// TIA Portal V17 export
// export: Created 2024-08-26T21:07:18.1732783Z, ExportSetting WithDefaults, DisplayName Totally Integrated Automation Portal, DisplayVersion V17 Update 7, DisplayName TIA Portal Openness, DisplayVersion V17 Update 7, DisplayName TIA Portal Version Control Interface, DisplayVersion V17, DisplayName SINAMICS Startdrive Advanced, DisplayVersion V17 SP2, DisplayName SINAMICS Startdrive G110M, G120, G120C, G120D, G120P, G115D, DisplayVersion V17 SP2, DisplayName SINAMICS Startdrive G130, G150, S120, S150, SINAMICS MV, S210, DisplayVersion V17 SP2, DisplayName STEP 7 Professional, DisplayVersion V17 Update 7, DisplayName STEP 7 Safety, DisplayVersion V17 Update 6, DisplayName WinCC Advanced / Unified PC, DisplayVersion V17 Update 7
FUNCTION "hmiControl" : Void   // FC3, LAD
{ S7_Optimized_Access := 'TRUE' }
VERSION : 0.1
// stored: AutoNumber true, IsIECCheckEnabled false, SetENOAutomatically false, UDAEnableTagReadback false
   VAR_TEMP   // added for the SCL form of the ladder/FBD networks
      _w1 : Bool;
      _w2 : Bool;
      _w3 : Bool;
      _w4 : Bool;
      _w5 : Bool;
      _w6 : Bool;
      _w7 : Bool;
      _w8 : Bool;
      _w9 : Bool;
      _w10 : Bool;
      _w11 : Bool;
      _w12 : Bool;
      _w13 : Bool;
      _w14 : Bool;
      _w15 : Bool;
      _w16 : Bool;
      _w17 : Bool;
      _w18 : Bool;
      _w19 : Bool;
      _w20 : Bool;
      _w21 : Bool;
      _w22 : Bool;
      _w23 : Bool;
      _w24 : Bool;
      _w25 : Bool;
      _w26 : Bool;
      _w27 : Bool;
      _w28 : Bool;
      _w29 : Bool;
      _w30 : Bool;
      _w31 : Bool;
      _w32 : Bool;
   END_VAR
BEGIN

REGION Network 1: VISUALIZACIÓN DE MODELOS: SI CADA MODELO TIENE UN NOMBRE GRABADO, SE ACTIVA SU VISUALIZACIÓN
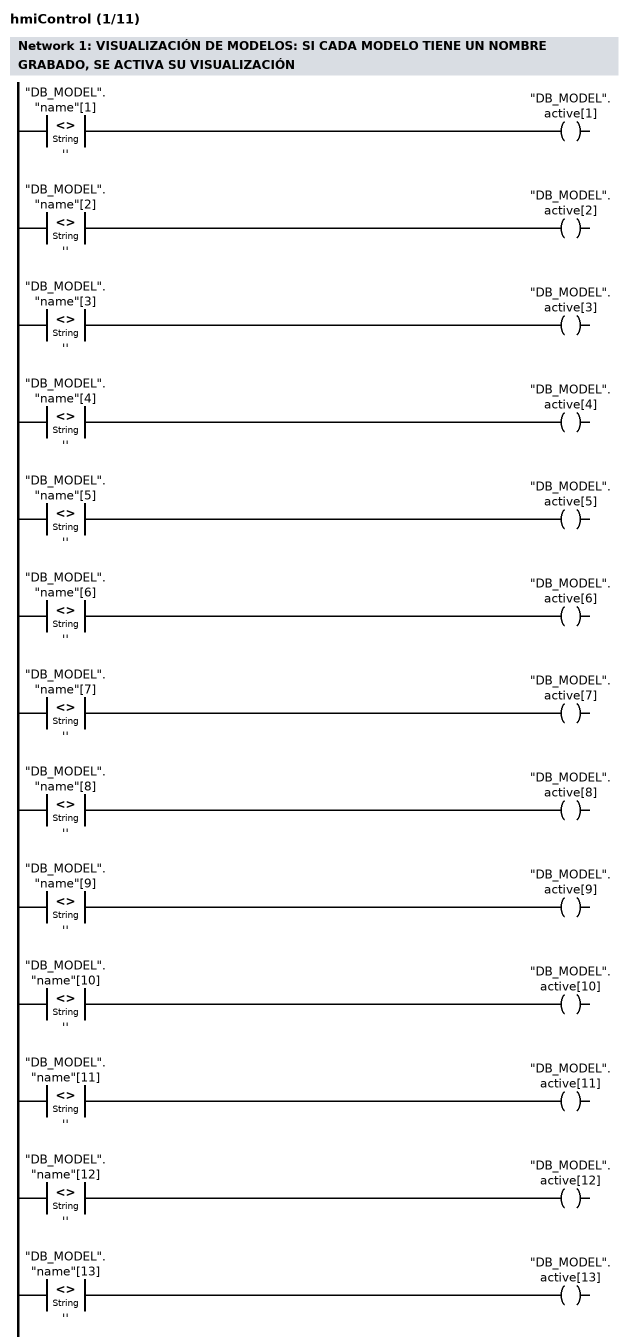
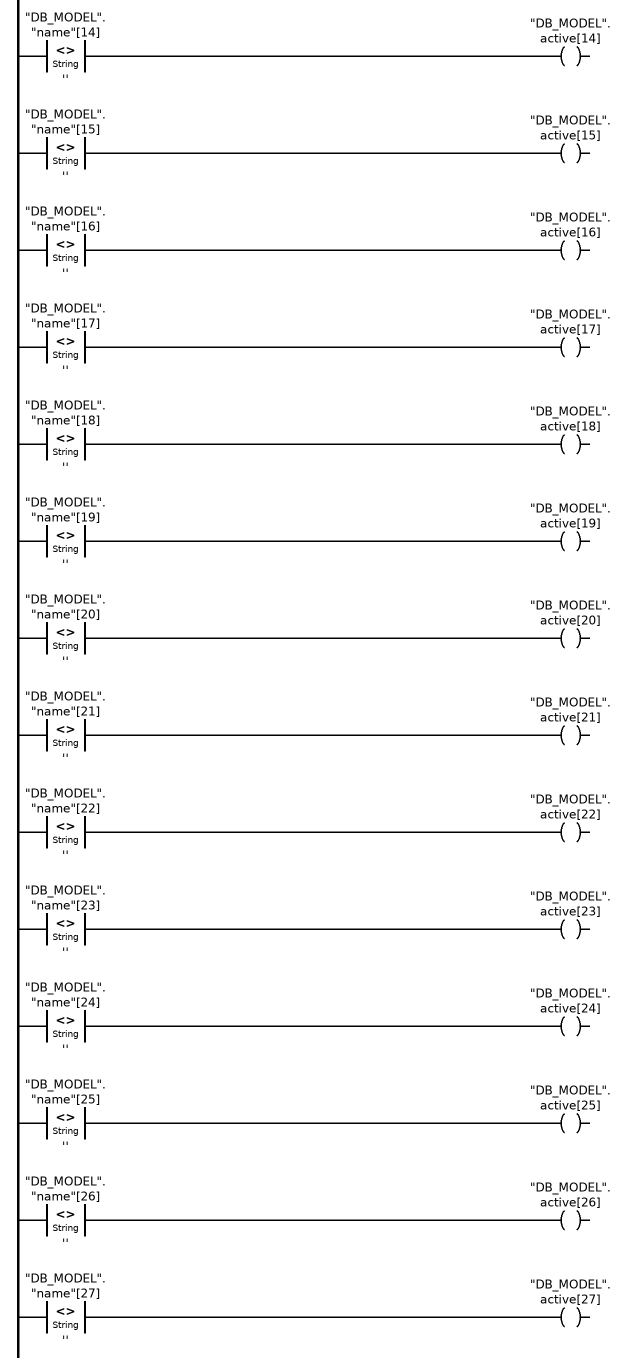
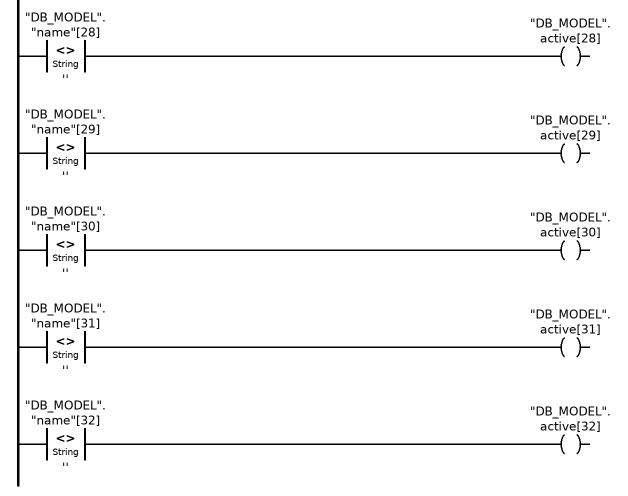
   RUNG wire#powerrail
      { S7_Templates := "SrcType := String" } NE_Contact(in1 := "DB_MODEL"."name"[1], in2 := '')
      Coil( "DB_MODEL".active[1] )
   END_RUNG
   RUNG wire#powerrail
      { S7_Templates := "SrcType := String" } NE_Contact(in1 := "DB_MODEL"."name"[2], in2 := '')
      Coil( "DB_MODEL".active[2] )
   END_RUNG
   RUNG wire#powerrail
      { S7_Templates := "SrcType := String" } NE_Contact(in1 := "DB_MODEL"."name"[3], in2 := '')
      Coil( "DB_MODEL".active[3] )
   END_RUNG
   RUNG wire#powerrail
      { S7_Templates := "SrcType := String" } NE_Contact(in1 := "DB_MODEL"."name"[4], in2 := '')
      Coil( "DB_MODEL".active[4] )
   END_RUNG
   RUNG wire#powerrail
      { S7_Templates := "SrcType := String" } NE_Contact(in1 := "DB_MODEL"."name"[5], in2 := '')
      Coil( "DB_MODEL".active[5] )
   END_RUNG
   RUNG wire#powerrail
      { S7_Templates := "SrcType := String" } NE_Contact(in1 := "DB_MODEL"."name"[6], in2 := '')
      Coil( "DB_MODEL".active[6] )
   END_RUNG
   RUNG wire#powerrail
      { S7_Templates := "SrcType := String" } NE_Contact(in1 := "DB_MODEL"."name"[7], in2 := '')
      Coil( "DB_MODEL".active[7] )
   END_RUNG
   RUNG wire#powerrail
      { S7_Templates := "SrcType := String" } NE_Contact(in1 := "DB_MODEL"."name"[8], in2 := '')
      Coil( "DB_MODEL".active[8] )
   END_RUNG
   RUNG wire#powerrail
      { S7_Templates := "SrcType := String" } NE_Contact(in1 := "DB_MODEL"."name"[9], in2 := '')
      Coil( "DB_MODEL".active[9] )
   END_RUNG
   RUNG wire#powerrail
      { S7_Templates := "SrcType := String" } NE_Contact(in1 := "DB_MODEL"."name"[10], in2 := '')
      Coil( "DB_MODEL".active[10] )
   END_RUNG
   RUNG wire#powerrail
      { S7_Templates := "SrcType := String" } NE_Contact(in1 := "DB_MODEL"."name"[11], in2 := '')
      Coil( "DB_MODEL".active[11] )
   END_RUNG
   RUNG wire#powerrail
      { S7_Templates := "SrcType := String" } NE_Contact(in1 := "DB_MODEL"."name"[12], in2 := '')
      Coil( "DB_MODEL".active[12] )
   END_RUNG
   RUNG wire#powerrail
      { S7_Templates := "SrcType := String" } NE_Contact(in1 := "DB_MODEL"."name"[13], in2 := '')
      Coil( "DB_MODEL".active[13] )
   END_RUNG
   RUNG wire#powerrail
      { S7_Templates := "SrcType := String" } NE_Contact(in1 := "DB_MODEL"."name"[14], in2 := '')
      Coil( "DB_MODEL".active[14] )
   END_RUNG
   RUNG wire#powerrail
      { S7_Templates := "SrcType := String" } NE_Contact(in1 := "DB_MODEL"."name"[15], in2 := '')
      Coil( "DB_MODEL".active[15] )
   END_RUNG
   RUNG wire#powerrail
      { S7_Templates := "SrcType := String" } NE_Contact(in1 := "DB_MODEL"."name"[16], in2 := '')
      Coil( "DB_MODEL".active[16] )
   END_RUNG
   RUNG wire#powerrail
      { S7_Templates := "SrcType := String" } NE_Contact(in1 := "DB_MODEL"."name"[17], in2 := '')
      Coil( "DB_MODEL".active[17] )
   END_RUNG
   RUNG wire#powerrail
      { S7_Templates := "SrcType := String" } NE_Contact(in1 := "DB_MODEL"."name"[18], in2 := '')
      Coil( "DB_MODEL".active[18] )
   END_RUNG
   RUNG wire#powerrail
      { S7_Templates := "SrcType := String" } NE_Contact(in1 := "DB_MODEL"."name"[19], in2 := '')
      Coil( "DB_MODEL".active[19] )
   END_RUNG
   RUNG wire#powerrail
      { S7_Templates := "SrcType := String" } NE_Contact(in1 := "DB_MODEL"."name"[20], in2 := '')
      Coil( "DB_MODEL".active[20] )
   END_RUNG
   RUNG wire#powerrail
      { S7_Templates := "SrcType := String" } NE_Contact(in1 := "DB_MODEL"."name"[21], in2 := '')
      Coil( "DB_MODEL".active[21] )
   END_RUNG
   RUNG wire#powerrail
      { S7_Templates := "SrcType := String" } NE_Contact(in1 := "DB_MODEL"."name"[22], in2 := '')
      Coil( "DB_MODEL".active[22] )
   END_RUNG
   RUNG wire#powerrail
      { S7_Templates := "SrcType := String" } NE_Contact(in1 := "DB_MODEL"."name"[23], in2 := '')
      Coil( "DB_MODEL".active[23] )
   END_RUNG
   RUNG wire#powerrail
      { S7_Templates := "SrcType := String" } NE_Contact(in1 := "DB_MODEL"."name"[24], in2 := '')
      Coil( "DB_MODEL".active[24] )
   END_RUNG
   RUNG wire#powerrail
      { S7_Templates := "SrcType := String" } NE_Contact(in1 := "DB_MODEL"."name"[25], in2 := '')
      Coil( "DB_MODEL".active[25] )
   END_RUNG
   RUNG wire#powerrail
      { S7_Templates := "SrcType := String" } NE_Contact(in1 := "DB_MODEL"."name"[26], in2 := '')
      Coil( "DB_MODEL".active[26] )
   END_RUNG
   RUNG wire#powerrail
      { S7_Templates := "SrcType := String" } NE_Contact(in1 := "DB_MODEL"."name"[27], in2 := '')
      Coil( "DB_MODEL".active[27] )
   END_RUNG
   RUNG wire#powerrail
      { S7_Templates := "SrcType := String" } NE_Contact(in1 := "DB_MODEL"."name"[28], in2 := '')
      Coil( "DB_MODEL".active[28] )
   END_RUNG
   RUNG wire#powerrail
      { S7_Templates := "SrcType := String" } NE_Contact(in1 := "DB_MODEL"."name"[29], in2 := '')
      Coil( "DB_MODEL".active[29] )
   END_RUNG
   RUNG wire#powerrail
      { S7_Templates := "SrcType := String" } NE_Contact(in1 := "DB_MODEL"."name"[30], in2 := '')
      Coil( "DB_MODEL".active[30] )
   END_RUNG
   RUNG wire#powerrail
      { S7_Templates := "SrcType := String" } NE_Contact(in1 := "DB_MODEL"."name"[31], in2 := '')
      Coil( "DB_MODEL".active[31] )
   END_RUNG
   RUNG wire#powerrail
      { S7_Templates := "SrcType := String" } NE_Contact(in1 := "DB_MODEL"."name"[32], in2 := '')
      Coil( "DB_MODEL".active[32] )
   END_RUNG
   // the same network as SCL:
   "DB_MODEL".active[1] := "DB_MODEL"."name"[1] <> '';
   "DB_MODEL".active[2] := "DB_MODEL"."name"[2] <> '';
   "DB_MODEL".active[3] := "DB_MODEL"."name"[3] <> '';
   "DB_MODEL".active[4] := "DB_MODEL"."name"[4] <> '';
   "DB_MODEL".active[5] := "DB_MODEL"."name"[5] <> '';
   "DB_MODEL".active[6] := "DB_MODEL"."name"[6] <> '';
   "DB_MODEL".active[7] := "DB_MODEL"."name"[7] <> '';
   "DB_MODEL".active[8] := "DB_MODEL"."name"[8] <> '';
   "DB_MODEL".active[9] := "DB_MODEL"."name"[9] <> '';
   "DB_MODEL".active[10] := "DB_MODEL"."name"[10] <> '';
   "DB_MODEL".active[11] := "DB_MODEL"."name"[11] <> '';
   "DB_MODEL".active[12] := "DB_MODEL"."name"[12] <> '';
   "DB_MODEL".active[13] := "DB_MODEL"."name"[13] <> '';
   "DB_MODEL".active[14] := "DB_MODEL"."name"[14] <> '';
   "DB_MODEL".active[15] := "DB_MODEL"."name"[15] <> '';
   "DB_MODEL".active[16] := "DB_MODEL"."name"[16] <> '';
   "DB_MODEL".active[17] := "DB_MODEL"."name"[17] <> '';
   "DB_MODEL".active[18] := "DB_MODEL"."name"[18] <> '';
   "DB_MODEL".active[19] := "DB_MODEL"."name"[19] <> '';
   "DB_MODEL".active[20] := "DB_MODEL"."name"[20] <> '';
   "DB_MODEL".active[21] := "DB_MODEL"."name"[21] <> '';
   "DB_MODEL".active[22] := "DB_MODEL"."name"[22] <> '';
   "DB_MODEL".active[23] := "DB_MODEL"."name"[23] <> '';
   "DB_MODEL".active[24] := "DB_MODEL"."name"[24] <> '';
   "DB_MODEL".active[25] := "DB_MODEL"."name"[25] <> '';
   "DB_MODEL".active[26] := "DB_MODEL"."name"[26] <> '';
   "DB_MODEL".active[27] := "DB_MODEL"."name"[27] <> '';
   "DB_MODEL".active[28] := "DB_MODEL"."name"[28] <> '';
   "DB_MODEL".active[29] := "DB_MODEL"."name"[29] <> '';
   "DB_MODEL".active[30] := "DB_MODEL"."name"[30] <> '';
   "DB_MODEL".active[31] := "DB_MODEL"."name"[31] <> '';
   "DB_MODEL".active[32] := "DB_MODEL"."name"[32] <> '';
END_REGION

REGION Network 2: CURRENT MODEL NAME SHOWN IN HMI
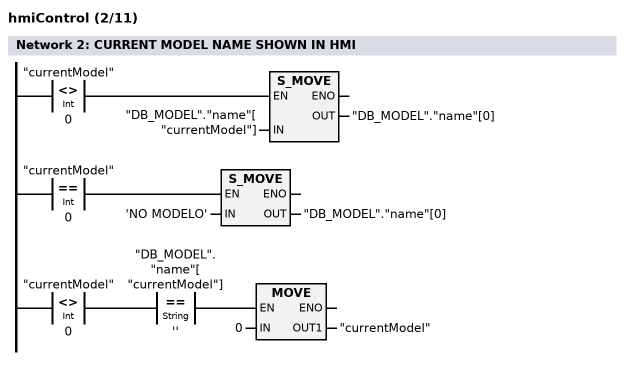
   RUNG wire#powerrail
      { S7_Templates := "SrcType := Int" } NE_Contact(in1 := "currentModel", in2 := 0)
      S_Move(in := "DB_MODEL"."name"["currentModel"], out => "DB_MODEL"."name"[0])
   END_RUNG
   RUNG wire#powerrail
      { S7_Templates := "SrcType := Int" } EQ_Contact(in1 := "currentModel", in2 := 0)
      S_Move(in := 'NO MODELO', out => "DB_MODEL"."name"[0])
   END_RUNG
   RUNG wire#powerrail
      { S7_Templates := "SrcType := Int" } NE_Contact(in1 := "currentModel", in2 := 0)
      { S7_Templates := "SrcType := String" } EQ_Contact(in1 := "DB_MODEL"."name"["currentModel"], in2 := '')
      Move(in := 0, out1 => "currentModel")
   END_RUNG
   // the same network as SCL:
   IF "currentModel" <> 0 THEN "DB_MODEL"."name"[0] := "DB_MODEL"."name"["currentModel"]; END_IF;
   IF "currentModel" = 0 THEN "DB_MODEL"."name"[0] := 'NO MODELO'; END_IF;
   IF ("currentModel" <> 0) AND ("DB_MODEL"."name"["currentModel"] = '') THEN "currentModel" := 0; END_IF;
END_REGION

REGION Network 3: MODEL CHANGE (VARIABLE ACTUALIZATION)
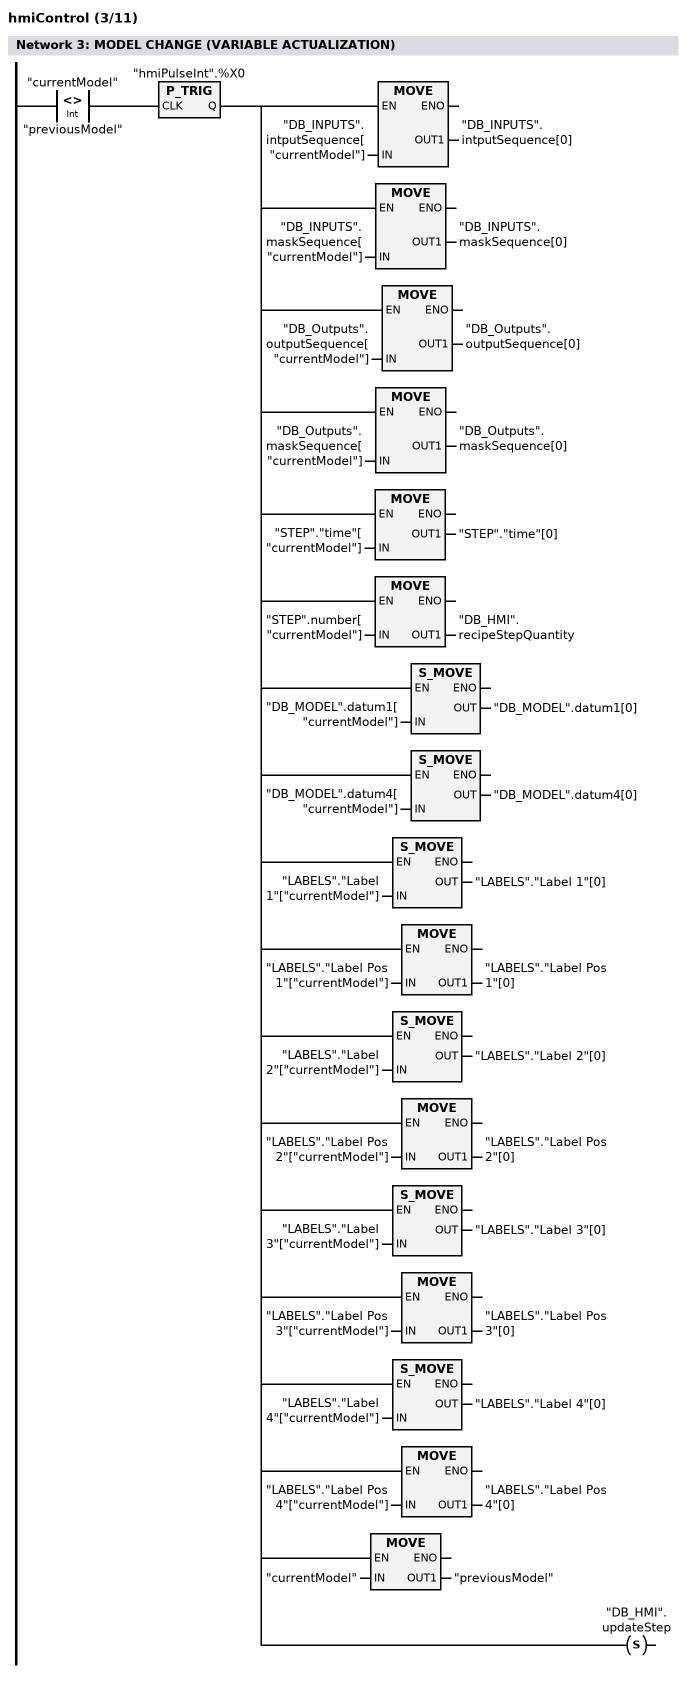
   RUNG wire#powerrail
      { S7_Templates := "SrcType := Int" } NE_Contact(in1 := "currentModel", in2 := "previousModel")
      P_Trig( "hmiPulseInt".%X0 )
      wire#w1
      Move(in := "DB_INPUTS".intputSequence["currentModel"], out1 => "DB_INPUTS".intputSequence[0])
   END_RUNG
   RUNG wire#w1
      Move(in := "DB_INPUTS".maskSequence["currentModel"], out1 => "DB_INPUTS".maskSequence[0])
   END_RUNG
   RUNG wire#w1
      Move(in := "DB_Outputs".outputSequence["currentModel"], out1 => "DB_Outputs".outputSequence[0])
   END_RUNG
   RUNG wire#w1
      Move(in := "DB_Outputs".maskSequence["currentModel"], out1 => "DB_Outputs".maskSequence[0])
   END_RUNG
   RUNG wire#w1
      Move(in := "STEP"."time"["currentModel"], out1 => "STEP"."time"[0])
   END_RUNG
   RUNG wire#w1
      Move(in := "STEP".number["currentModel"], out1 => "DB_HMI".recipeStepQuantity)
   END_RUNG
   RUNG wire#w1
      S_Move(in := "DB_MODEL".datum1["currentModel"], out => "DB_MODEL".datum1[0])
   END_RUNG
   RUNG wire#w1
      S_Move(in := "DB_MODEL".datum4["currentModel"], out => "DB_MODEL".datum4[0])
   END_RUNG
   RUNG wire#w1
      S_Move(in := "LABELS"."Label 1"["currentModel"], out => "LABELS"."Label 1"[0])
   END_RUNG
   RUNG wire#w1
      Move(in := "LABELS"."Label Pos 1"["currentModel"], out1 => "LABELS"."Label Pos 1"[0])
   END_RUNG
   RUNG wire#w1
      S_Move(in := "LABELS"."Label 2"["currentModel"], out => "LABELS"."Label 2"[0])
   END_RUNG
   RUNG wire#w1
      Move(in := "LABELS"."Label Pos 2"["currentModel"], out1 => "LABELS"."Label Pos 2"[0])
   END_RUNG
   RUNG wire#w1
      S_Move(in := "LABELS"."Label 3"["currentModel"], out => "LABELS"."Label 3"[0])
   END_RUNG
   RUNG wire#w1
      Move(in := "LABELS"."Label Pos 3"["currentModel"], out1 => "LABELS"."Label Pos 3"[0])
   END_RUNG
   RUNG wire#w1
      S_Move(in := "LABELS"."Label 4"["currentModel"], out => "LABELS"."Label 4"[0])
   END_RUNG
   RUNG wire#w1
      Move(in := "LABELS"."Label Pos 4"["currentModel"], out1 => "LABELS"."Label Pos 4"[0])
   END_RUNG
   RUNG wire#w1
      Move(in := "currentModel", out1 => "previousModel")
   END_RUNG
   RUNG wire#w1
      S_Coil( "DB_HMI".updateStep )
   END_RUNG
   // the same network as SCL:
   #_w1 := "currentModel" <> "previousModel";
   #_w2 := #_w1 AND NOT "hmiPulseInt".%X0;   // rising edge
   "hmiPulseInt".%X0 := #_w1;
   IF #_w2 THEN
       "DB_INPUTS".intputSequence[0] := "DB_INPUTS".intputSequence["currentModel"];
       "DB_INPUTS".maskSequence[0] := "DB_INPUTS".maskSequence["currentModel"];
       "DB_Outputs".outputSequence[0] := "DB_Outputs".outputSequence["currentModel"];
       "DB_Outputs".maskSequence[0] := "DB_Outputs".maskSequence["currentModel"];
       "STEP"."time"[0] := "STEP"."time"["currentModel"];
       "DB_HMI".recipeStepQuantity := "STEP".number["currentModel"];
       "DB_MODEL".datum1[0] := "DB_MODEL".datum1["currentModel"];
       "DB_MODEL".datum4[0] := "DB_MODEL".datum4["currentModel"];
       "LABELS"."Label 1"[0] := "LABELS"."Label 1"["currentModel"];
       "LABELS"."Label Pos 1"[0] := "LABELS"."Label Pos 1"["currentModel"];
       "LABELS"."Label 2"[0] := "LABELS"."Label 2"["currentModel"];
       "LABELS"."Label Pos 2"[0] := "LABELS"."Label Pos 2"["currentModel"];
       "LABELS"."Label 3"[0] := "LABELS"."Label 3"["currentModel"];
       "LABELS"."Label Pos 3"[0] := "LABELS"."Label Pos 3"["currentModel"];
       "LABELS"."Label 4"[0] := "LABELS"."Label 4"["currentModel"];
       "LABELS"."Label Pos 4"[0] := "LABELS"."Label Pos 4"["currentModel"];
       "previousModel" := "currentModel";
       "DB_HMI".updateStep := TRUE;
   END_IF;
END_REGION

REGION Network 4: STEP CHANGE IN RECIPE
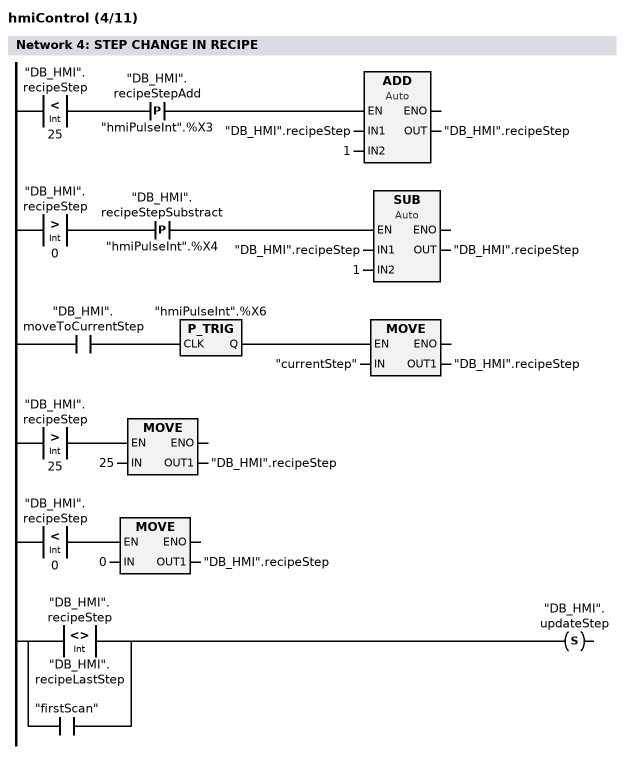
   RUNG wire#powerrail
      { S7_Templates := "SrcType := Int" } LT_Contact(in1 := "DB_HMI".recipeStep, in2 := 25)
      P_Contact(operand := "DB_HMI".recipeStepAdd, bit := "hmiPulseInt".%X3)
      Add(in1 := "DB_HMI".recipeStep, in2 := 1, out => "DB_HMI".recipeStep)
   END_RUNG
   RUNG wire#powerrail
      { S7_Templates := "SrcType := Int" } GT_Contact(in1 := "DB_HMI".recipeStep, in2 := 0)
      P_Contact(operand := "DB_HMI".recipeStepSubstract, bit := "hmiPulseInt".%X4)
      Sub(in1 := "DB_HMI".recipeStep, in2 := 1, out => "DB_HMI".recipeStep)
   END_RUNG
   RUNG wire#powerrail
      Contact( "DB_HMI".moveToCurrentStep )
      P_Trig( "hmiPulseInt".%X6 )
      Move(in := "currentStep", out1 => "DB_HMI".recipeStep)
   END_RUNG
   RUNG wire#powerrail
      { S7_Templates := "SrcType := Int" } GT_Contact(in1 := "DB_HMI".recipeStep, in2 := 25)
      Move(in := 25, out1 => "DB_HMI".recipeStep)
   END_RUNG
   RUNG wire#powerrail
      { S7_Templates := "SrcType := Int" } LT_Contact(in1 := "DB_HMI".recipeStep, in2 := 0)
      Move(in := 0, out1 => "DB_HMI".recipeStep)
   END_RUNG
   RUNG wire#powerrail
      { S7_Templates := "SrcType := Int" } NE_Contact(in1 := "DB_HMI".recipeStep, in2 := "DB_HMI".recipeLastStep)
      wire#w1
      S_Coil( "DB_HMI".updateStep )
   END_RUNG
   RUNG wire#powerrail
      Contact( "firstScan" )
   END_RUNG wire#w1
   // the same network as SCL:
   #_w1 := ("DB_HMI".recipeStep < 25) AND "DB_HMI".recipeStepAdd AND NOT "hmiPulseInt".%X3;   // rising edge of "DB_HMI".recipeStepAdd
   "hmiPulseInt".%X3 := "DB_HMI".recipeStepAdd;
   IF #_w1 THEN "DB_HMI".recipeStep := "DB_HMI".recipeStep + 1; END_IF;
   #_w2 := ("DB_HMI".recipeStep > 0) AND "DB_HMI".recipeStepSubstract AND NOT "hmiPulseInt".%X4;   // rising edge of "DB_HMI".recipeStepSubstract
   "hmiPulseInt".%X4 := "DB_HMI".recipeStepSubstract;
   IF #_w2 THEN "DB_HMI".recipeStep := "DB_HMI".recipeStep - 1; END_IF;
   #_w3 := "DB_HMI".moveToCurrentStep AND NOT "hmiPulseInt".%X6;   // rising edge
   "hmiPulseInt".%X6 := "DB_HMI".moveToCurrentStep;
   IF #_w3 THEN "DB_HMI".recipeStep := "currentStep"; END_IF;
   IF "DB_HMI".recipeStep > 25 THEN "DB_HMI".recipeStep := 25; END_IF;
   IF "DB_HMI".recipeStep < 0 THEN "DB_HMI".recipeStep := 0; END_IF;
   IF ("DB_HMI".recipeStep <> "DB_HMI".recipeLastStep) OR "firstScan" THEN
       "DB_HMI".updateStep := TRUE;
   END_IF;
END_REGION

REGION Network 5: HMI PARAMETER REFRESH FROM STEP CHANGE
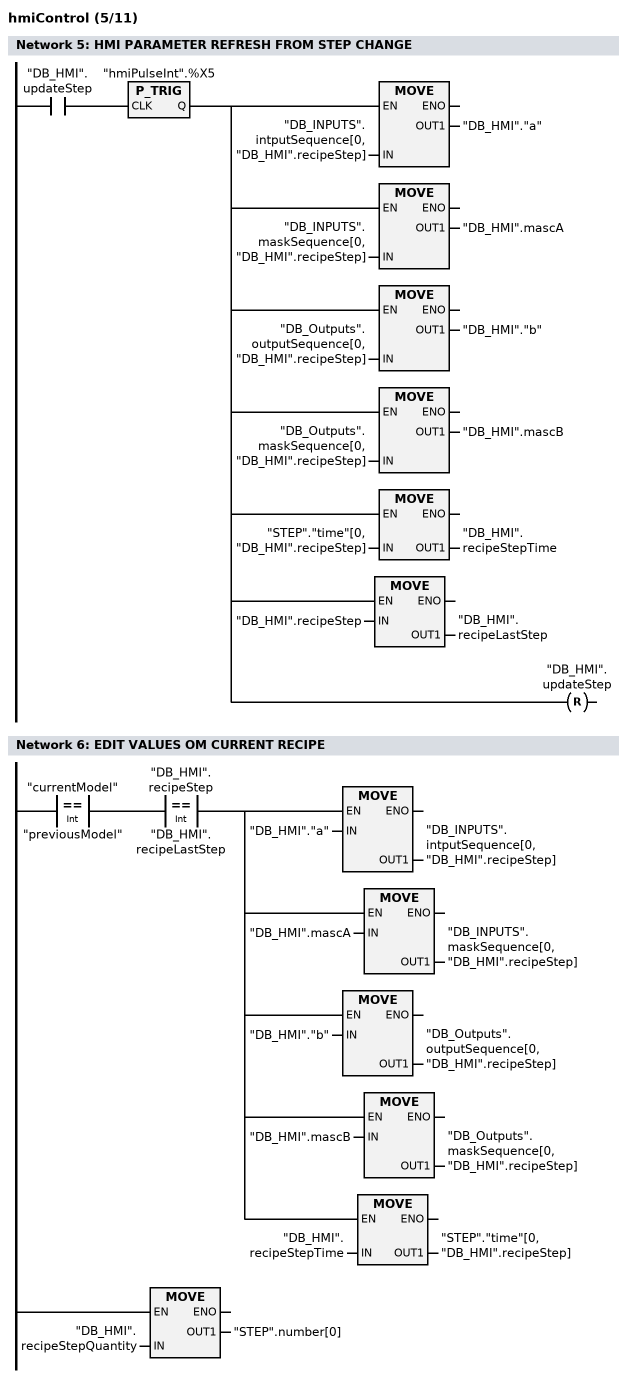
   RUNG wire#powerrail
      Contact( "DB_HMI".updateStep )
      P_Trig( "hmiPulseInt".%X5 )
      wire#w1
      Move(in := "DB_INPUTS".intputSequence[0, "DB_HMI".recipeStep], out1 => "DB_HMI"."a")
   END_RUNG
   RUNG wire#w1
      Move(in := "DB_INPUTS".maskSequence[0, "DB_HMI".recipeStep], out1 => "DB_HMI".mascA)
   END_RUNG
   RUNG wire#w1
      Move(in := "DB_Outputs".outputSequence[0, "DB_HMI".recipeStep], out1 => "DB_HMI"."b")
   END_RUNG
   RUNG wire#w1
      Move(in := "DB_Outputs".maskSequence[0, "DB_HMI".recipeStep], out1 => "DB_HMI".mascB)
   END_RUNG
   RUNG wire#w1
      Move(in := "STEP"."time"[0, "DB_HMI".recipeStep], out1 => "DB_HMI".recipeStepTime)
   END_RUNG
   RUNG wire#w1
      Move(in := "DB_HMI".recipeStep, out1 => "DB_HMI".recipeLastStep)
   END_RUNG
   RUNG wire#w1
      R_Coil( "DB_HMI".updateStep )
   END_RUNG
   // the same network as SCL:
   #_w1 := "DB_HMI".updateStep AND NOT "hmiPulseInt".%X5;   // rising edge
   "hmiPulseInt".%X5 := "DB_HMI".updateStep;
   IF #_w1 THEN
       "DB_HMI"."a" := "DB_INPUTS".intputSequence[0, "DB_HMI".recipeStep];
       "DB_HMI".mascA := "DB_INPUTS".maskSequence[0, "DB_HMI".recipeStep];
       "DB_HMI"."b" := "DB_Outputs".outputSequence[0, "DB_HMI".recipeStep];
       "DB_HMI".mascB := "DB_Outputs".maskSequence[0, "DB_HMI".recipeStep];
       "DB_HMI".recipeStepTime := "STEP"."time"[0, "DB_HMI".recipeStep];
       "DB_HMI".recipeLastStep := "DB_HMI".recipeStep;
       "DB_HMI".updateStep := FALSE;
   END_IF;
END_REGION

REGION Network 6: EDIT VALUES OM CURRENT RECIPE
   RUNG wire#powerrail
      { S7_Templates := "SrcType := Int" } EQ_Contact(in1 := "currentModel", in2 := "previousModel")
      { S7_Templates := "SrcType := Int" } EQ_Contact(in1 := "DB_HMI".recipeStep, in2 := "DB_HMI".recipeLastStep)
      wire#w1
      Move(in := "DB_HMI"."a", out1 => "DB_INPUTS".intputSequence[0, "DB_HMI".recipeStep])
   END_RUNG
   RUNG wire#w1
      Move(in := "DB_HMI".mascA, out1 => "DB_INPUTS".maskSequence[0, "DB_HMI".recipeStep])
   END_RUNG
   RUNG wire#w1
      Move(in := "DB_HMI"."b", out1 => "DB_Outputs".outputSequence[0, "DB_HMI".recipeStep])
   END_RUNG
   RUNG wire#w1
      Move(in := "DB_HMI".mascB, out1 => "DB_Outputs".maskSequence[0, "DB_HMI".recipeStep])
   END_RUNG
   RUNG wire#w1
      Move(in := "DB_HMI".recipeStepTime, out1 => "STEP"."time"[0, "DB_HMI".recipeStep])
   END_RUNG
   RUNG wire#powerrail
      Move(in := "DB_HMI".recipeStepQuantity, out1 => "STEP".number[0])
   END_RUNG
   // the same network as SCL:
   #_w1 := ("currentModel" = "previousModel") AND ("DB_HMI".recipeStep = "DB_HMI".recipeLastStep);
   IF #_w1 THEN
       "DB_INPUTS".intputSequence[0, "DB_HMI".recipeStep] := "DB_HMI"."a";
       "DB_INPUTS".maskSequence[0, "DB_HMI".recipeStep] := "DB_HMI".mascA;
       "DB_Outputs".outputSequence[0, "DB_HMI".recipeStep] := "DB_HMI"."b";
       "DB_Outputs".maskSequence[0, "DB_HMI".recipeStep] := "DB_HMI".mascB;
       "STEP"."time"[0, "DB_HMI".recipeStep] := "DB_HMI".recipeStepTime;
   END_IF;
   "STEP".number[0] := "DB_HMI".recipeStepQuantity;
END_REGION

REGION Network 7: WRITE AND READN IN SCREEN
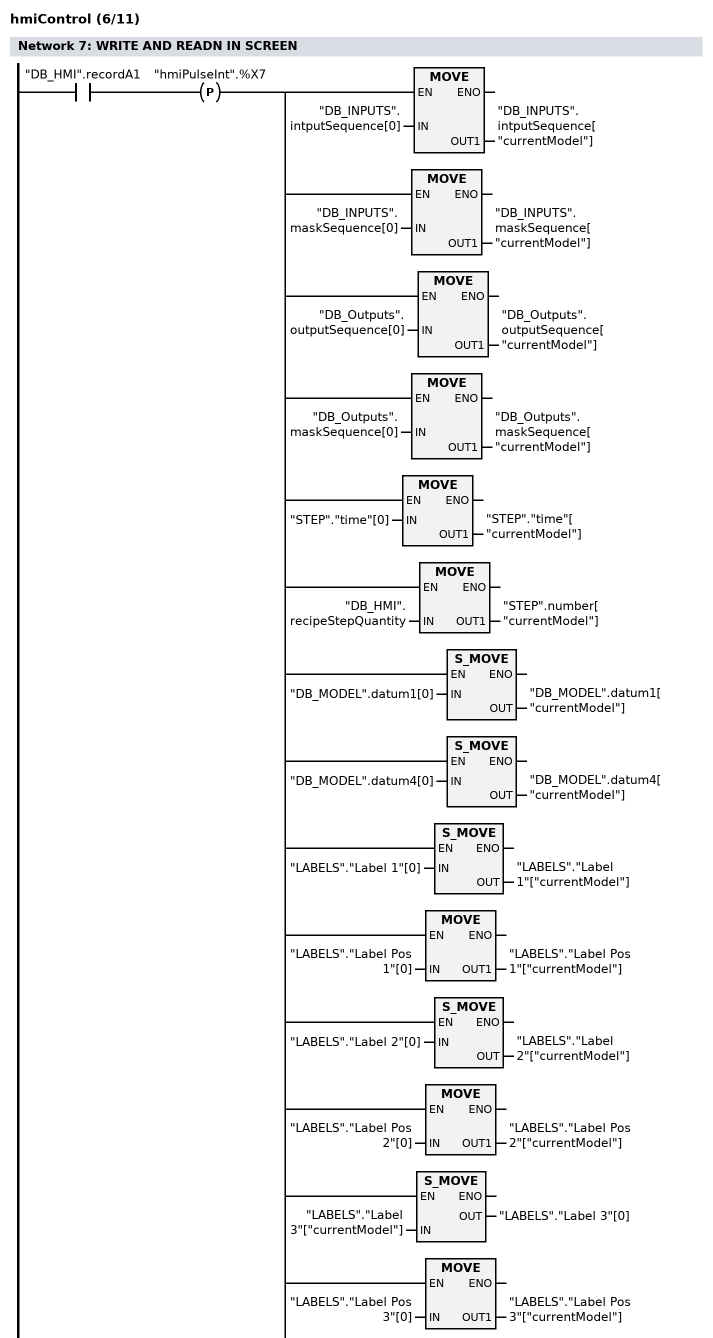
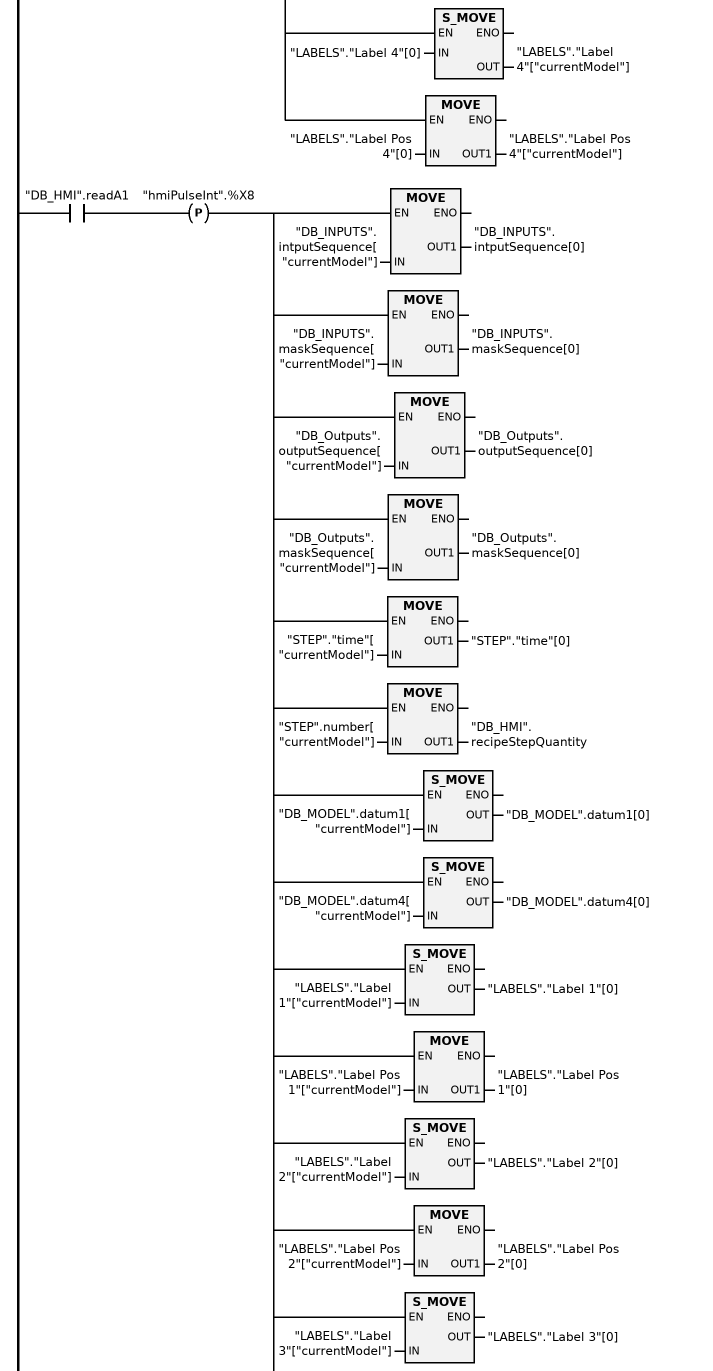
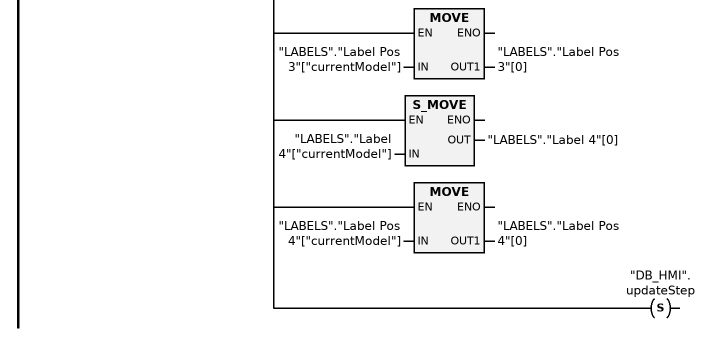
   RUNG wire#powerrail
      Contact( "DB_HMI".recordA1 )
      P_Trig( "hmiPulseInt".%X7 )
      wire#w1
      Move(in := "DB_INPUTS".intputSequence[0], out1 => "DB_INPUTS".intputSequence["currentModel"])
   END_RUNG
   RUNG wire#w1
      Move(in := "DB_INPUTS".maskSequence[0], out1 => "DB_INPUTS".maskSequence["currentModel"])
   END_RUNG
   RUNG wire#w1
      Move(in := "DB_Outputs".outputSequence[0], out1 => "DB_Outputs".outputSequence["currentModel"])
   END_RUNG
   RUNG wire#w1
      Move(in := "DB_Outputs".maskSequence[0], out1 => "DB_Outputs".maskSequence["currentModel"])
   END_RUNG
   RUNG wire#w1
      Move(in := "STEP"."time"[0], out1 => "STEP"."time"["currentModel"])
   END_RUNG
   RUNG wire#w1
      Move(in := "DB_HMI".recipeStepQuantity, out1 => "STEP".number["currentModel"])
   END_RUNG
   RUNG wire#w1
      S_Move(in := "DB_MODEL".datum1[0], out => "DB_MODEL".datum1["currentModel"])
   END_RUNG
   RUNG wire#w1
      S_Move(in := "DB_MODEL".datum4[0], out => "DB_MODEL".datum4["currentModel"])
   END_RUNG
   RUNG wire#w1
      S_Move(in := "LABELS"."Label 1"[0], out => "LABELS"."Label 1"["currentModel"])
   END_RUNG
   RUNG wire#w1
      Move(in := "LABELS"."Label Pos 1"[0], out1 => "LABELS"."Label Pos 1"["currentModel"])
   END_RUNG
   RUNG wire#w1
      S_Move(in := "LABELS"."Label 2"[0], out => "LABELS"."Label 2"["currentModel"])
   END_RUNG
   RUNG wire#w1
      Move(in := "LABELS"."Label Pos 2"[0], out1 => "LABELS"."Label Pos 2"["currentModel"])
   END_RUNG
   RUNG wire#w1
      S_Move(in := "LABELS"."Label 3"["currentModel"], out => "LABELS"."Label 3"[0])
   END_RUNG
   RUNG wire#w1
      Move(in := "LABELS"."Label Pos 3"[0], out1 => "LABELS"."Label Pos 3"["currentModel"])
   END_RUNG
   RUNG wire#w1
      S_Move(in := "LABELS"."Label 4"[0], out => "LABELS"."Label 4"["currentModel"])
   END_RUNG
   RUNG wire#w1
      Move(in := "LABELS"."Label Pos 4"[0], out1 => "LABELS"."Label Pos 4"["currentModel"])
   END_RUNG
   RUNG wire#powerrail
      Contact( "DB_HMI".readA1 )
      P_Trig( "hmiPulseInt".%X8 )
      wire#w2
      Move(in := "DB_INPUTS".intputSequence["currentModel"], out1 => "DB_INPUTS".intputSequence[0])
   END_RUNG
   RUNG wire#w2
      Move(in := "DB_INPUTS".maskSequence["currentModel"], out1 => "DB_INPUTS".maskSequence[0])
   END_RUNG
   RUNG wire#w2
      Move(in := "DB_Outputs".outputSequence["currentModel"], out1 => "DB_Outputs".outputSequence[0])
   END_RUNG
   RUNG wire#w2
      Move(in := "DB_Outputs".maskSequence["currentModel"], out1 => "DB_Outputs".maskSequence[0])
   END_RUNG
   RUNG wire#w2
      Move(in := "STEP"."time"["currentModel"], out1 => "STEP"."time"[0])
   END_RUNG
   RUNG wire#w2
      Move(in := "STEP".number["currentModel"], out1 => "DB_HMI".recipeStepQuantity)
   END_RUNG
   RUNG wire#w2
      S_Move(in := "DB_MODEL".datum1["currentModel"], out => "DB_MODEL".datum1[0])
   END_RUNG
   RUNG wire#w2
      S_Move(in := "DB_MODEL".datum4["currentModel"], out => "DB_MODEL".datum4[0])
   END_RUNG
   RUNG wire#w2
      S_Move(in := "LABELS"."Label 1"["currentModel"], out => "LABELS"."Label 1"[0])
   END_RUNG
   RUNG wire#w2
      Move(in := "LABELS"."Label Pos 1"["currentModel"], out1 => "LABELS"."Label Pos 1"[0])
   END_RUNG
   RUNG wire#w2
      S_Move(in := "LABELS"."Label 2"["currentModel"], out => "LABELS"."Label 2"[0])
   END_RUNG
   RUNG wire#w2
      Move(in := "LABELS"."Label Pos 2"["currentModel"], out1 => "LABELS"."Label Pos 2"[0])
   END_RUNG
   RUNG wire#w2
      S_Move(in := "LABELS"."Label 3"["currentModel"], out => "LABELS"."Label 3"[0])
   END_RUNG
   RUNG wire#w2
      Move(in := "LABELS"."Label Pos 3"["currentModel"], out1 => "LABELS"."Label Pos 3"[0])
   END_RUNG
   RUNG wire#w2
      S_Move(in := "LABELS"."Label 4"["currentModel"], out => "LABELS"."Label 4"[0])
   END_RUNG
   RUNG wire#w2
      Move(in := "LABELS"."Label Pos 4"["currentModel"], out1 => "LABELS"."Label Pos 4"[0])
   END_RUNG
   RUNG wire#w2
      S_Coil( "DB_HMI".updateStep )
   END_RUNG
   // the same network as SCL:
   #_w1 := "DB_HMI".recordA1 AND NOT "hmiPulseInt".%X7;   // rising edge
   "hmiPulseInt".%X7 := "DB_HMI".recordA1;
   IF #_w1 THEN
       "DB_INPUTS".intputSequence["currentModel"] := "DB_INPUTS".intputSequence[0];
       "DB_INPUTS".maskSequence["currentModel"] := "DB_INPUTS".maskSequence[0];
       "DB_Outputs".outputSequence["currentModel"] := "DB_Outputs".outputSequence[0];
       "DB_Outputs".maskSequence["currentModel"] := "DB_Outputs".maskSequence[0];
       "STEP"."time"["currentModel"] := "STEP"."time"[0];
       "STEP".number["currentModel"] := "DB_HMI".recipeStepQuantity;
       "DB_MODEL".datum1["currentModel"] := "DB_MODEL".datum1[0];
       "DB_MODEL".datum4["currentModel"] := "DB_MODEL".datum4[0];
       "LABELS"."Label 1"["currentModel"] := "LABELS"."Label 1"[0];
       "LABELS"."Label Pos 1"["currentModel"] := "LABELS"."Label Pos 1"[0];
       "LABELS"."Label 2"["currentModel"] := "LABELS"."Label 2"[0];
       "LABELS"."Label Pos 2"["currentModel"] := "LABELS"."Label Pos 2"[0];
       "LABELS"."Label 3"[0] := "LABELS"."Label 3"["currentModel"];
       "LABELS"."Label Pos 3"["currentModel"] := "LABELS"."Label Pos 3"[0];
       "LABELS"."Label 4"["currentModel"] := "LABELS"."Label 4"[0];
       "LABELS"."Label Pos 4"["currentModel"] := "LABELS"."Label Pos 4"[0];
   END_IF;
   #_w2 := "DB_HMI".readA1 AND NOT "hmiPulseInt".%X8;   // rising edge
   "hmiPulseInt".%X8 := "DB_HMI".readA1;
   IF #_w2 THEN
       "DB_INPUTS".intputSequence[0] := "DB_INPUTS".intputSequence["currentModel"];
       "DB_INPUTS".maskSequence[0] := "DB_INPUTS".maskSequence["currentModel"];
       "DB_Outputs".outputSequence[0] := "DB_Outputs".outputSequence["currentModel"];
       "DB_Outputs".maskSequence[0] := "DB_Outputs".maskSequence["currentModel"];
       "STEP"."time"[0] := "STEP"."time"["currentModel"];
       "DB_HMI".recipeStepQuantity := "STEP".number["currentModel"];
       "DB_MODEL".datum1[0] := "DB_MODEL".datum1["currentModel"];
       "DB_MODEL".datum4[0] := "DB_MODEL".datum4["currentModel"];
       "LABELS"."Label 1"[0] := "LABELS"."Label 1"["currentModel"];
       "LABELS"."Label Pos 1"[0] := "LABELS"."Label Pos 1"["currentModel"];
       "LABELS"."Label 2"[0] := "LABELS"."Label 2"["currentModel"];
       "LABELS"."Label Pos 2"[0] := "LABELS"."Label Pos 2"["currentModel"];
       "LABELS"."Label 3"[0] := "LABELS"."Label 3"["currentModel"];
       "LABELS"."Label Pos 3"[0] := "LABELS"."Label Pos 3"["currentModel"];
       "LABELS"."Label 4"[0] := "LABELS"."Label 4"["currentModel"];
       "LABELS"."Label Pos 4"[0] := "LABELS"."Label Pos 4"["currentModel"];
       "DB_HMI".updateStep := TRUE;
   END_IF;
END_REGION

REGION Network 8: NUMBERS OF STEPS OF RECIPE
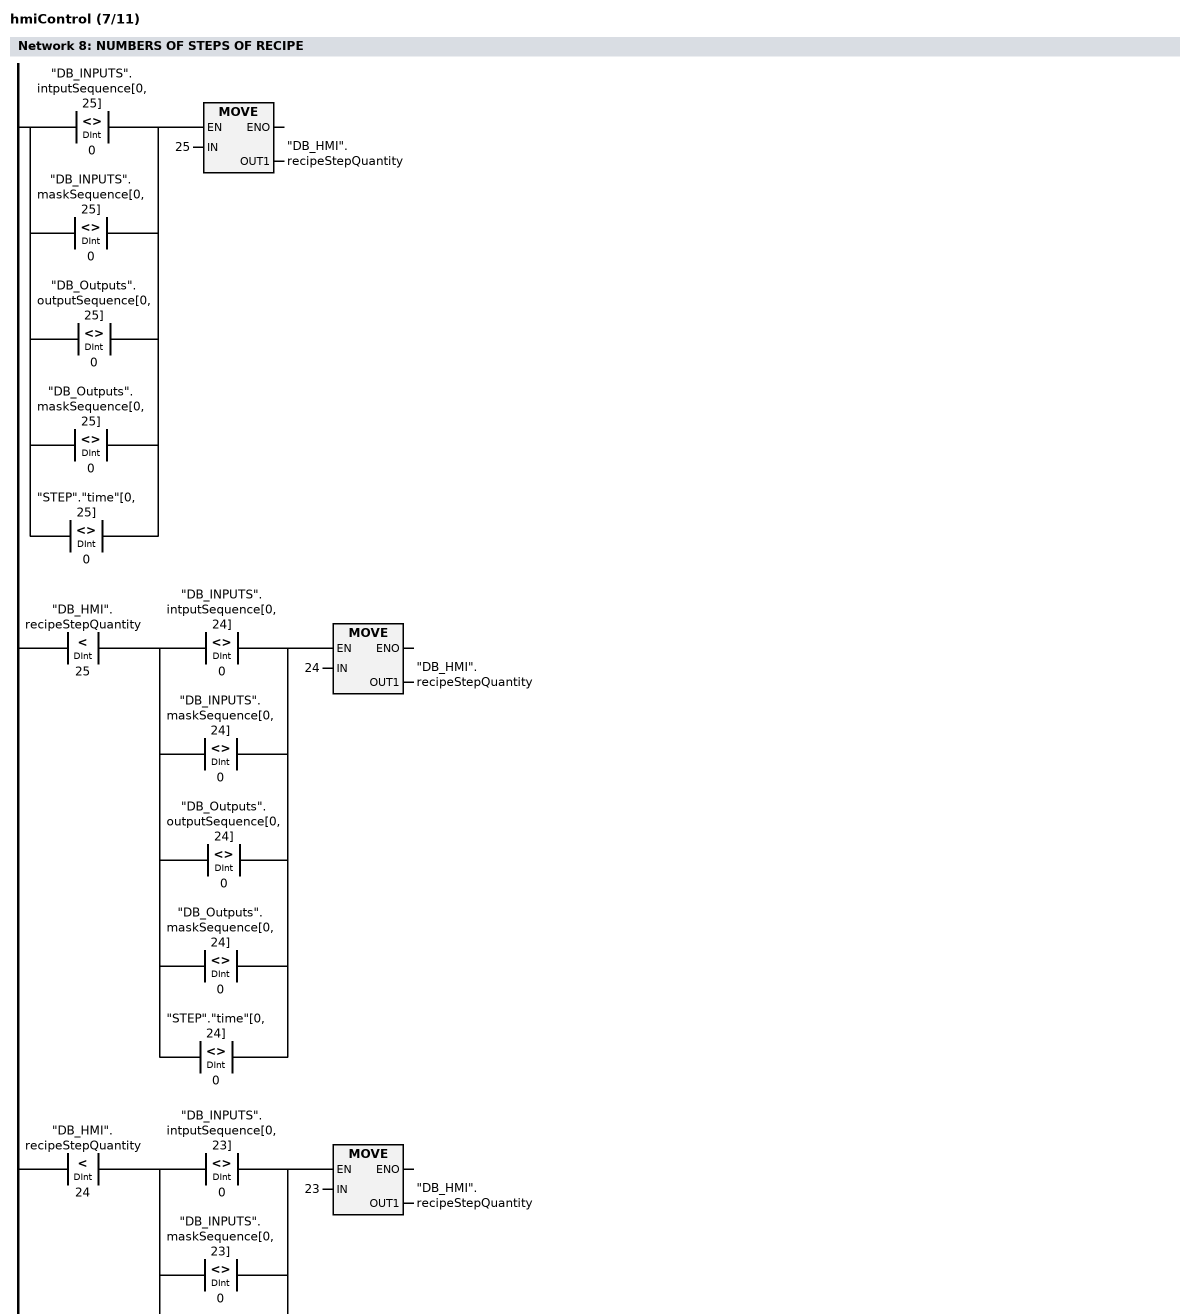
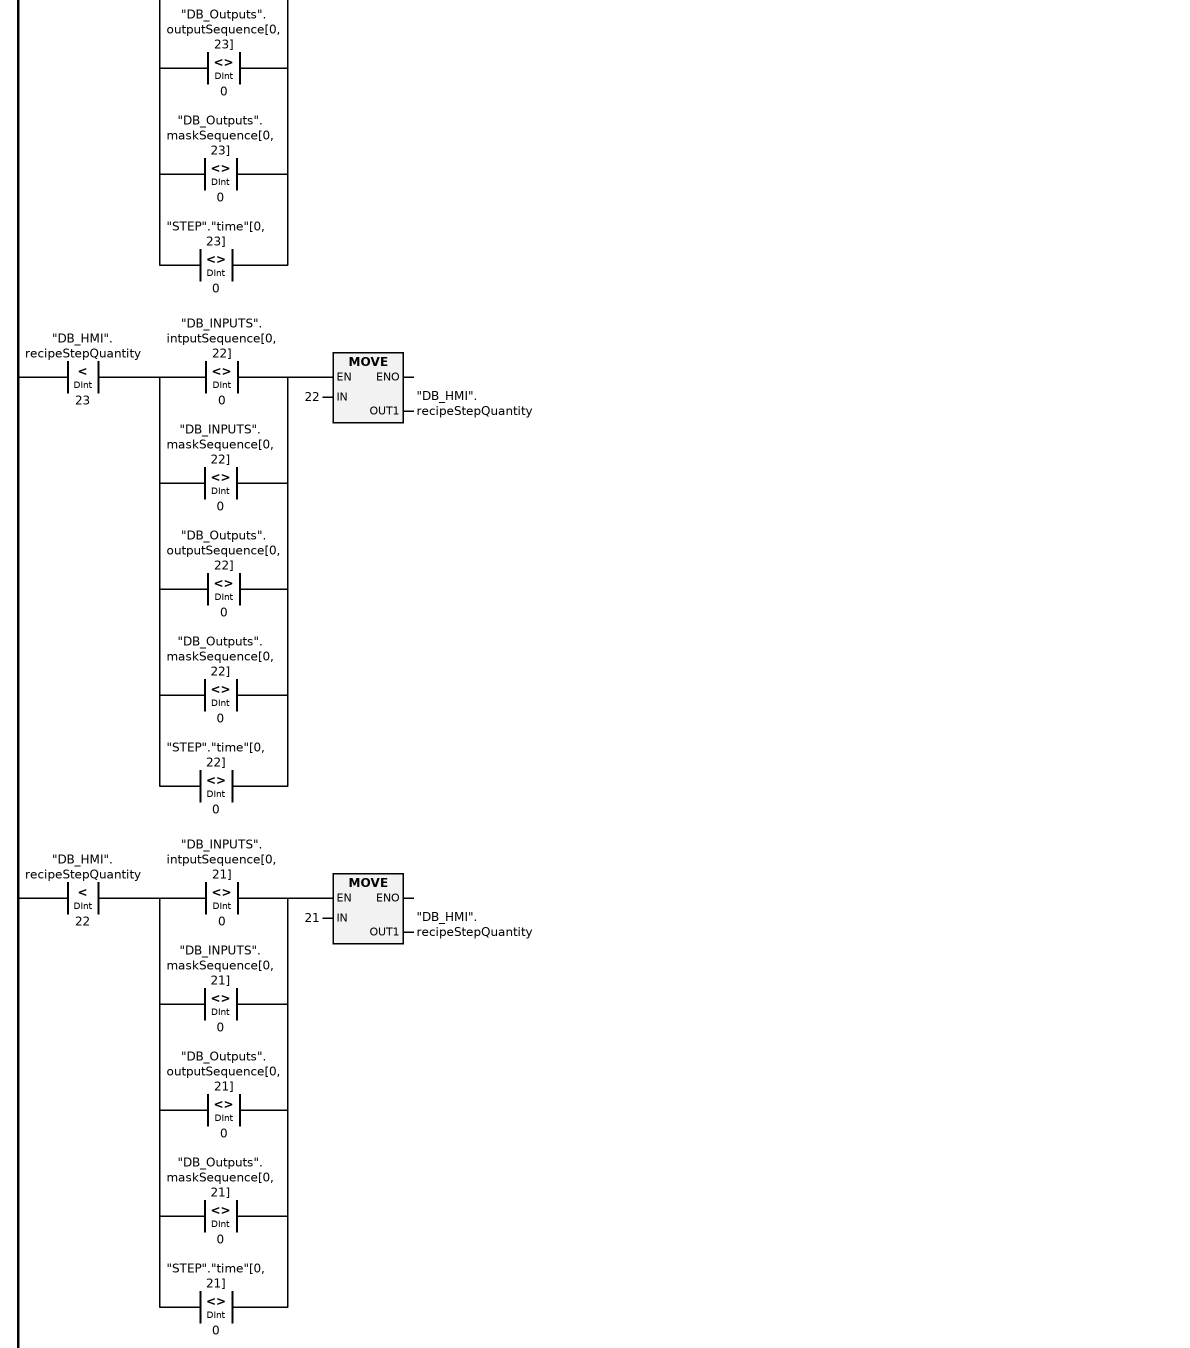
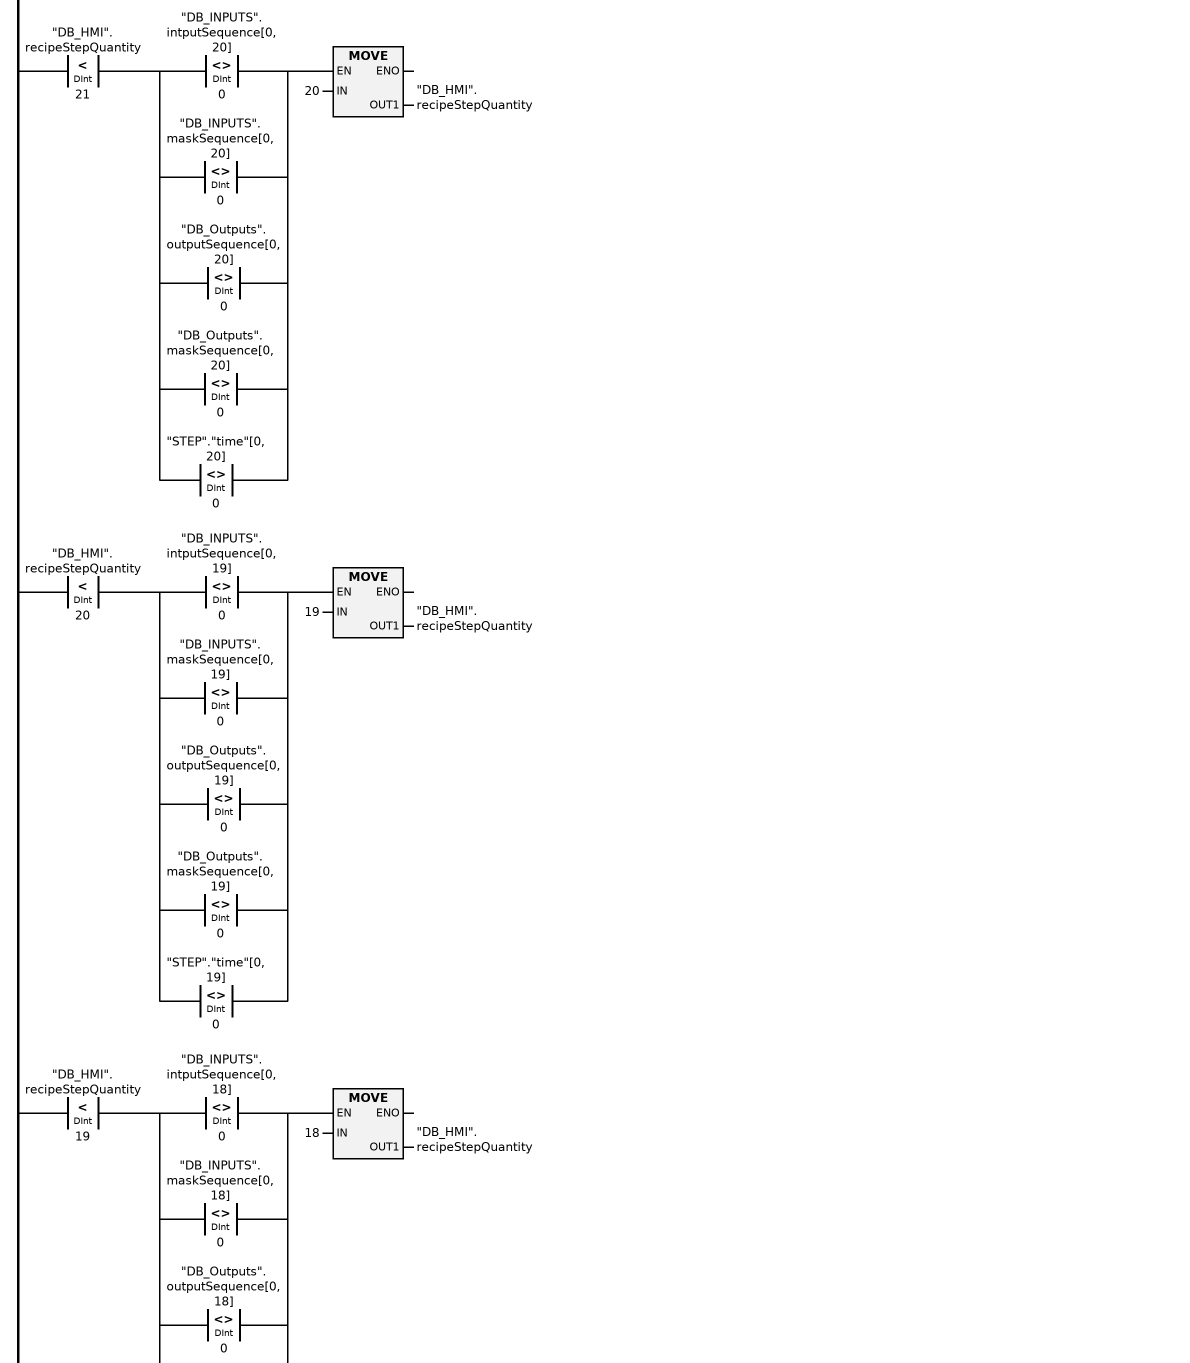
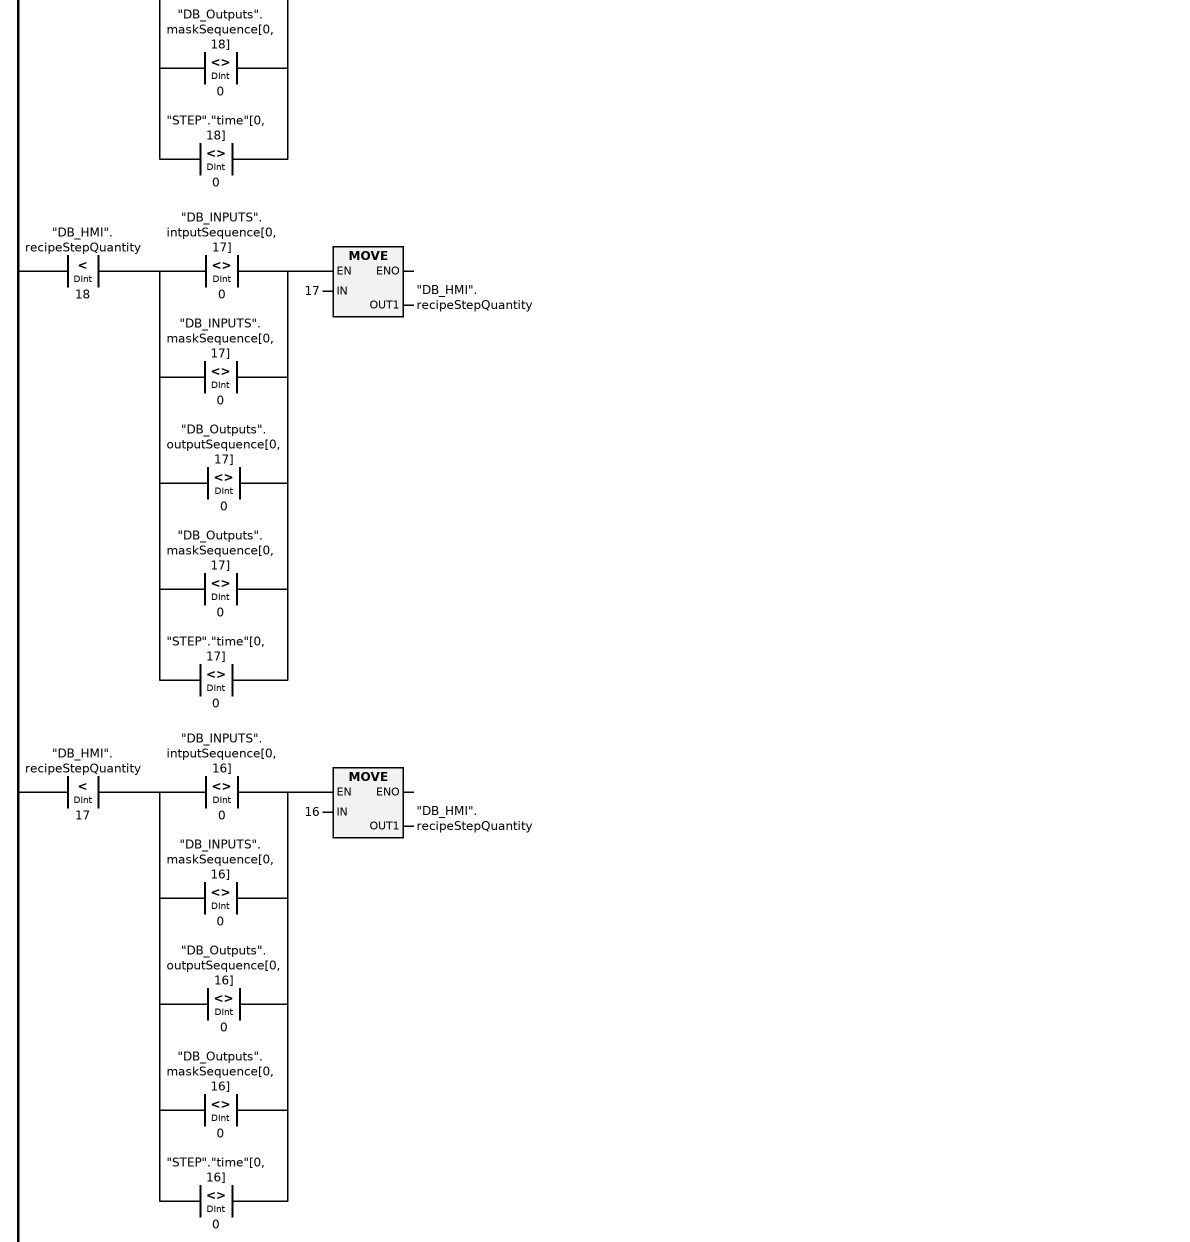
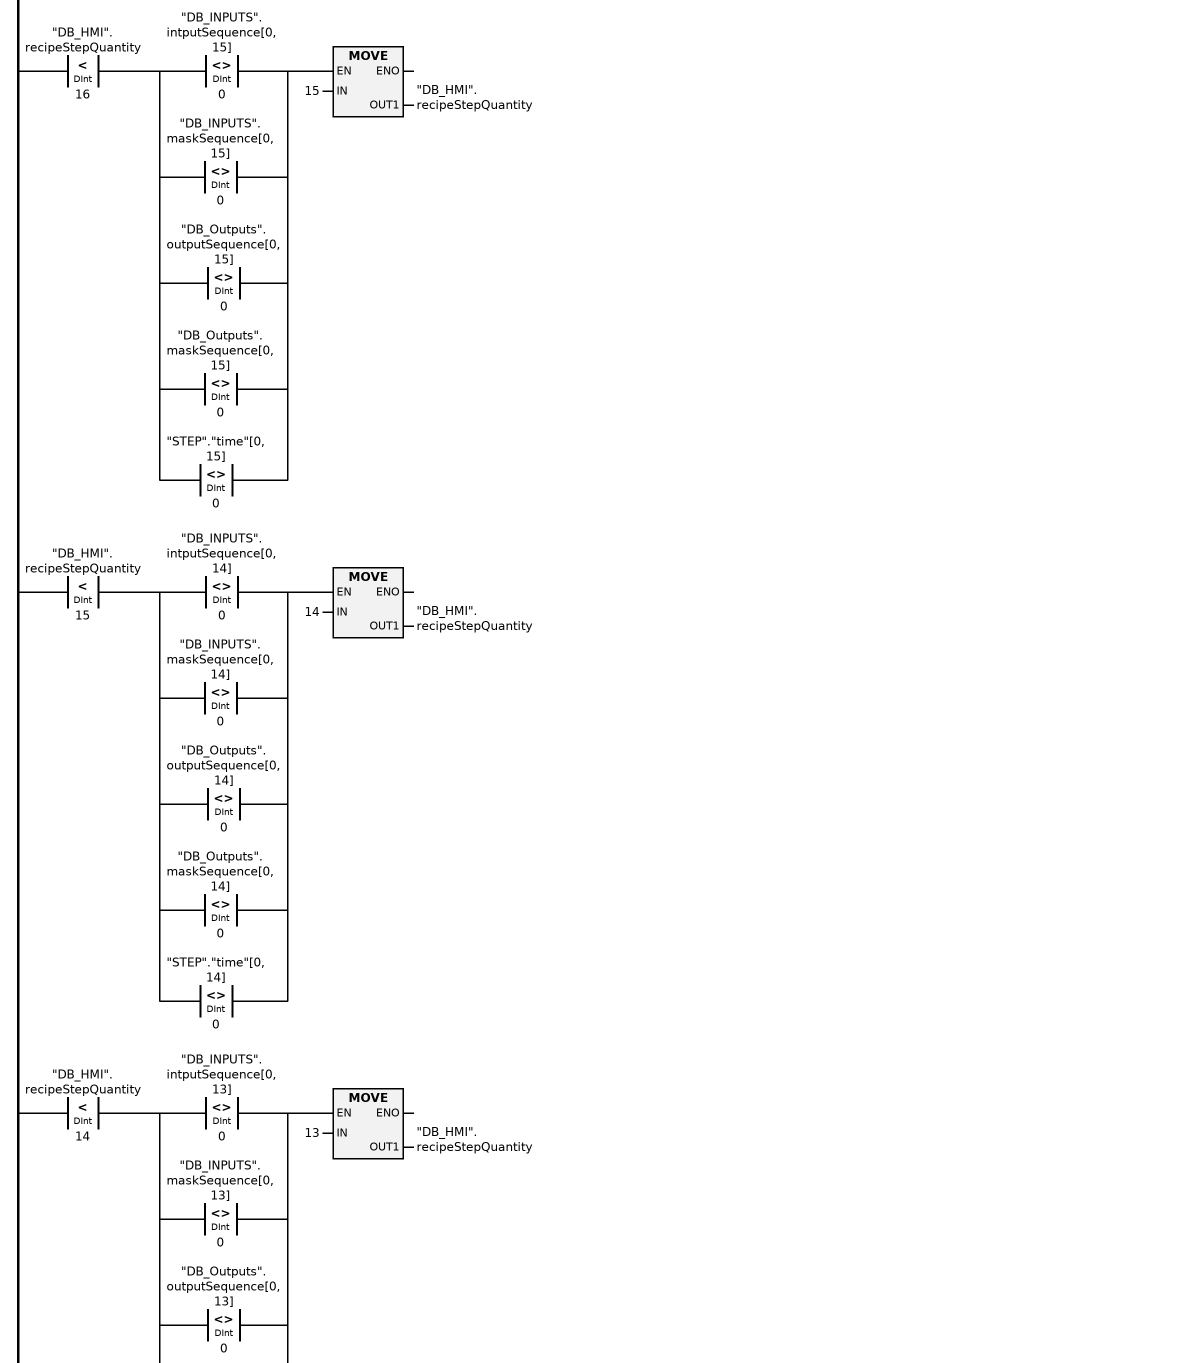
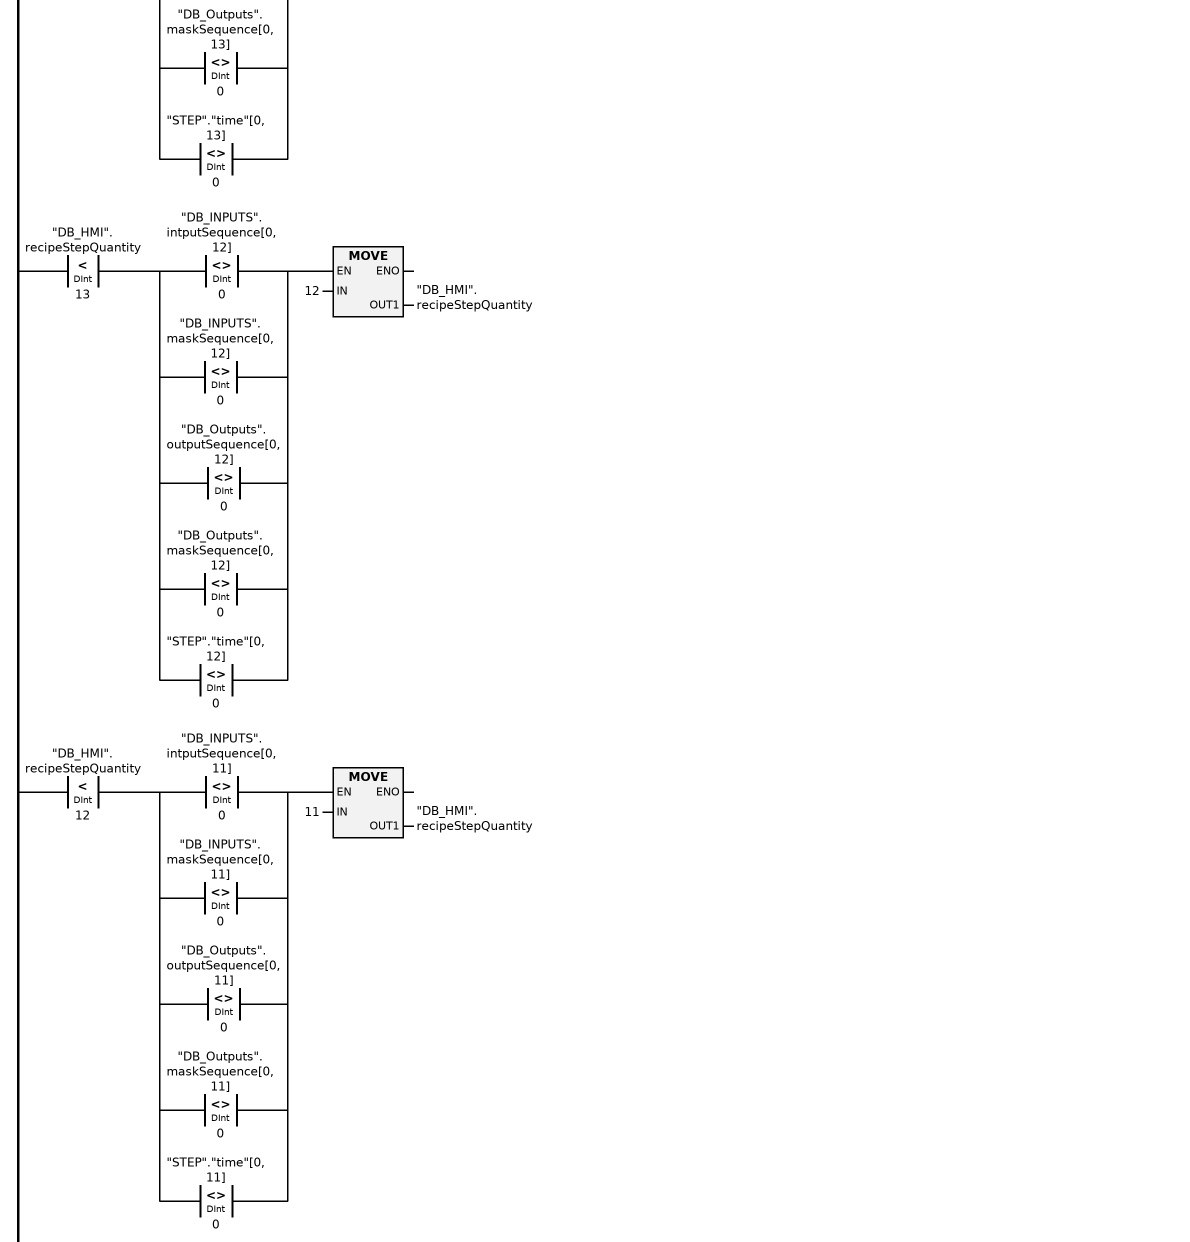
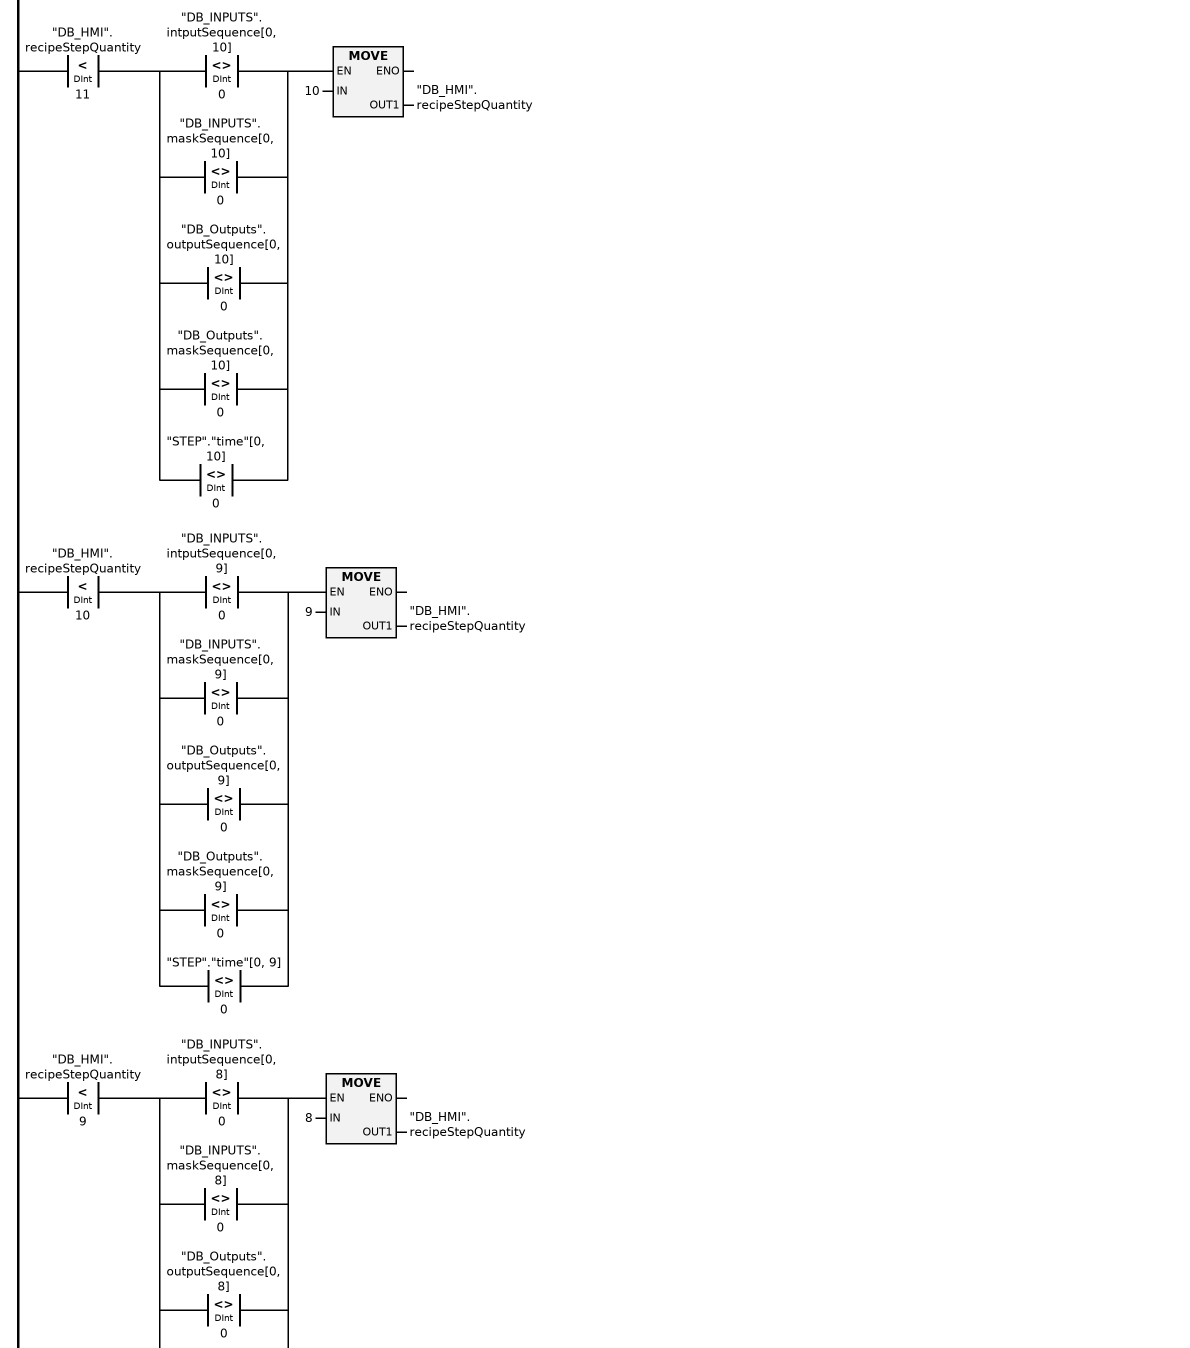
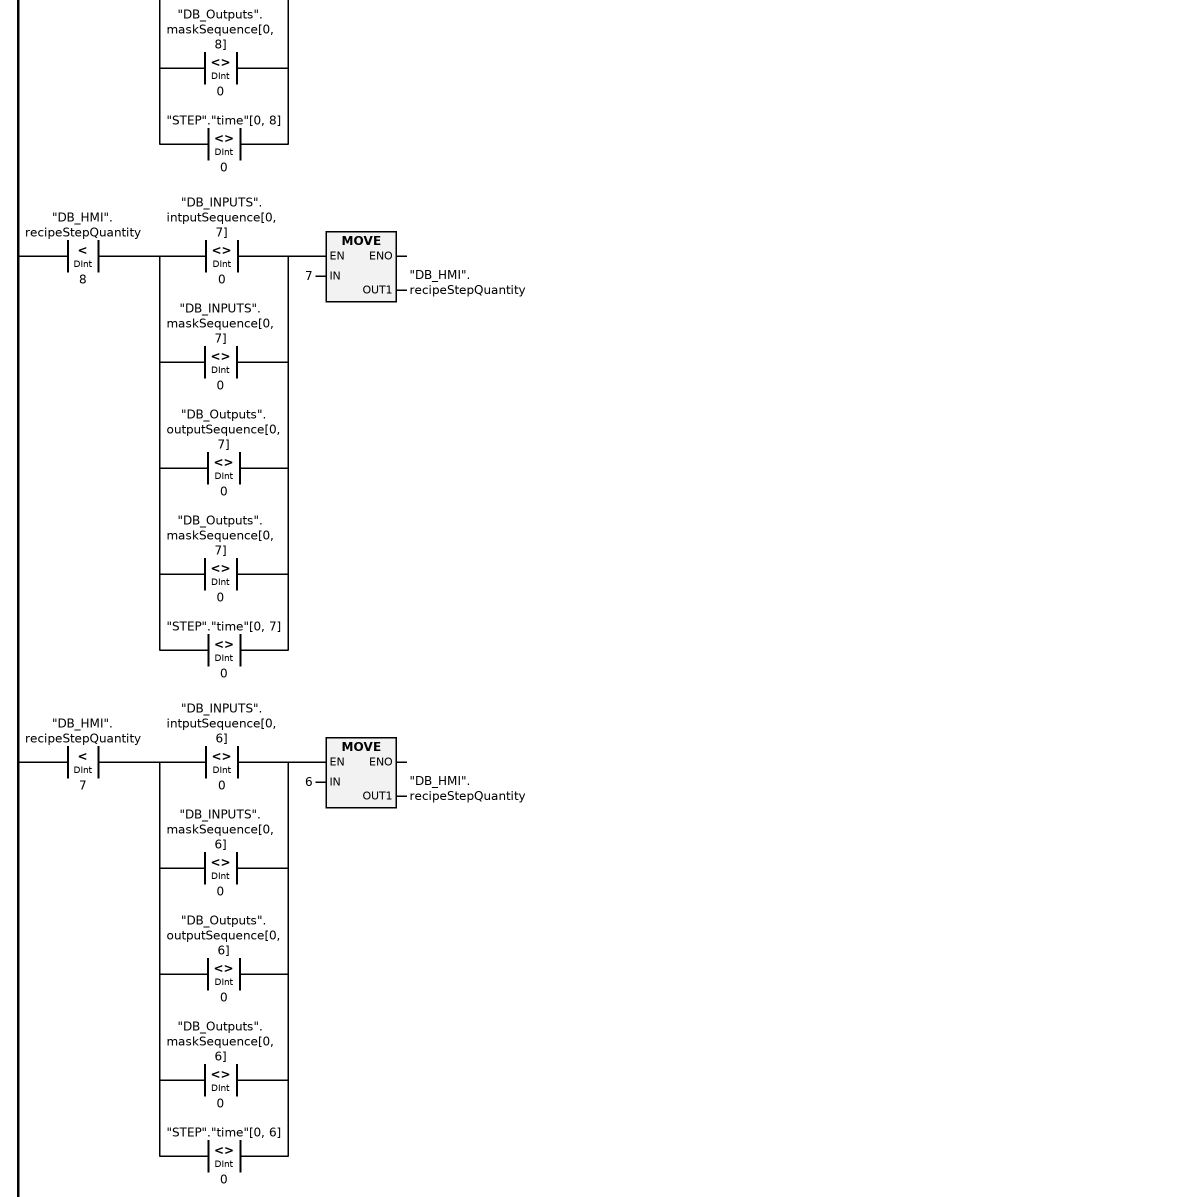
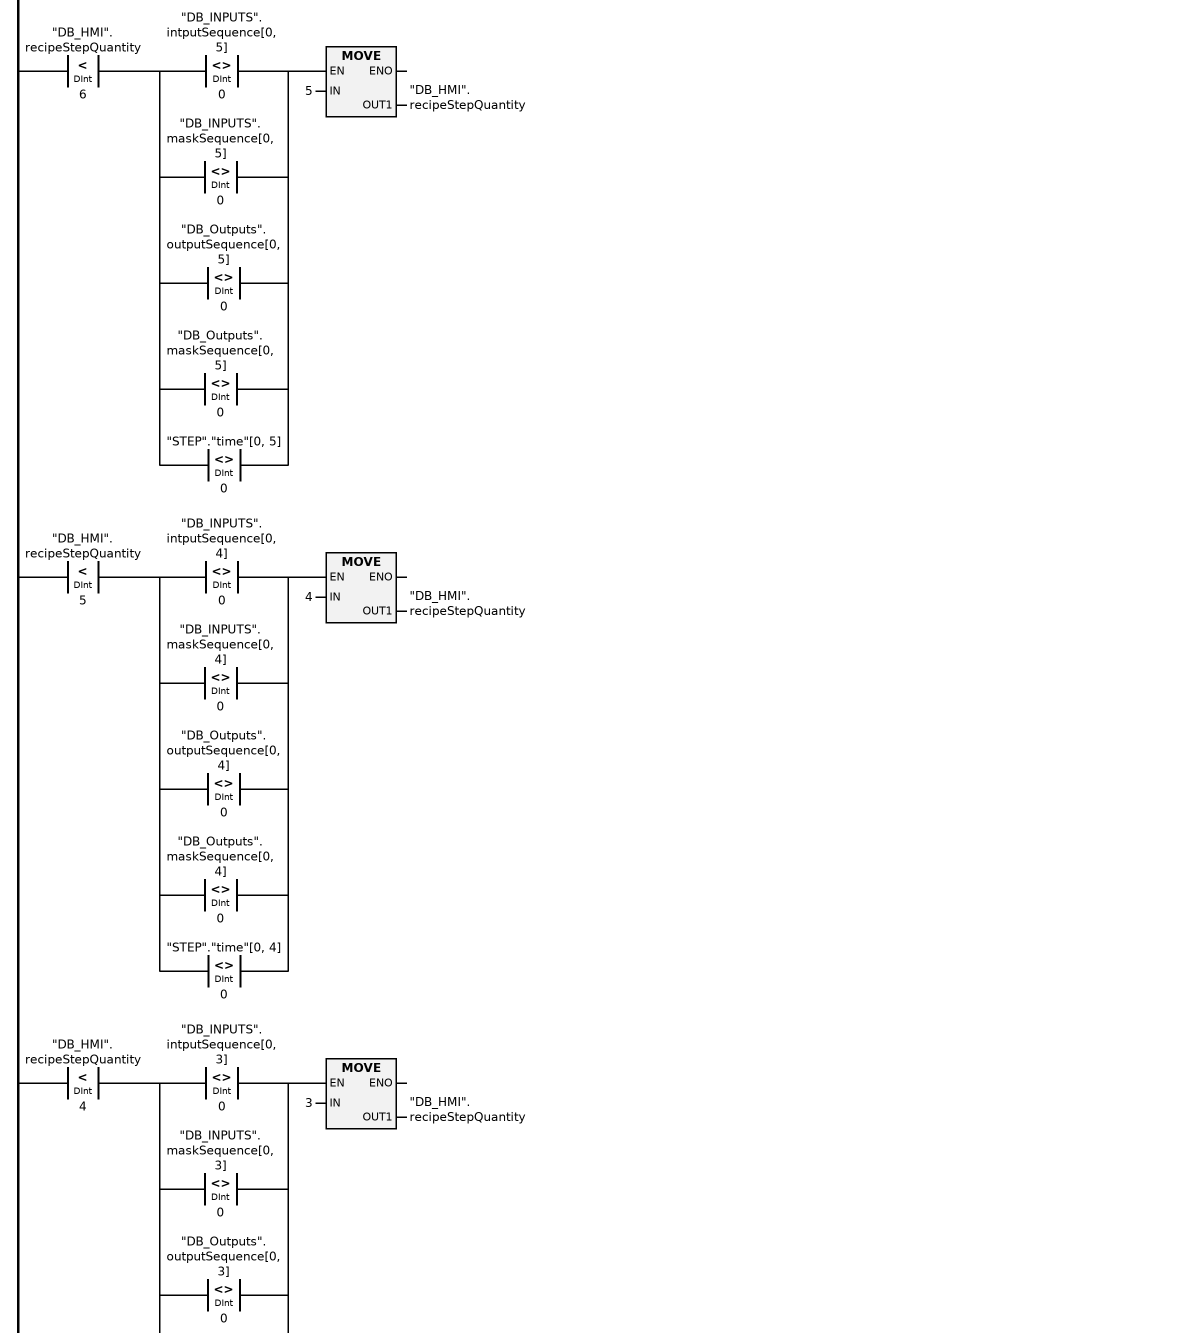
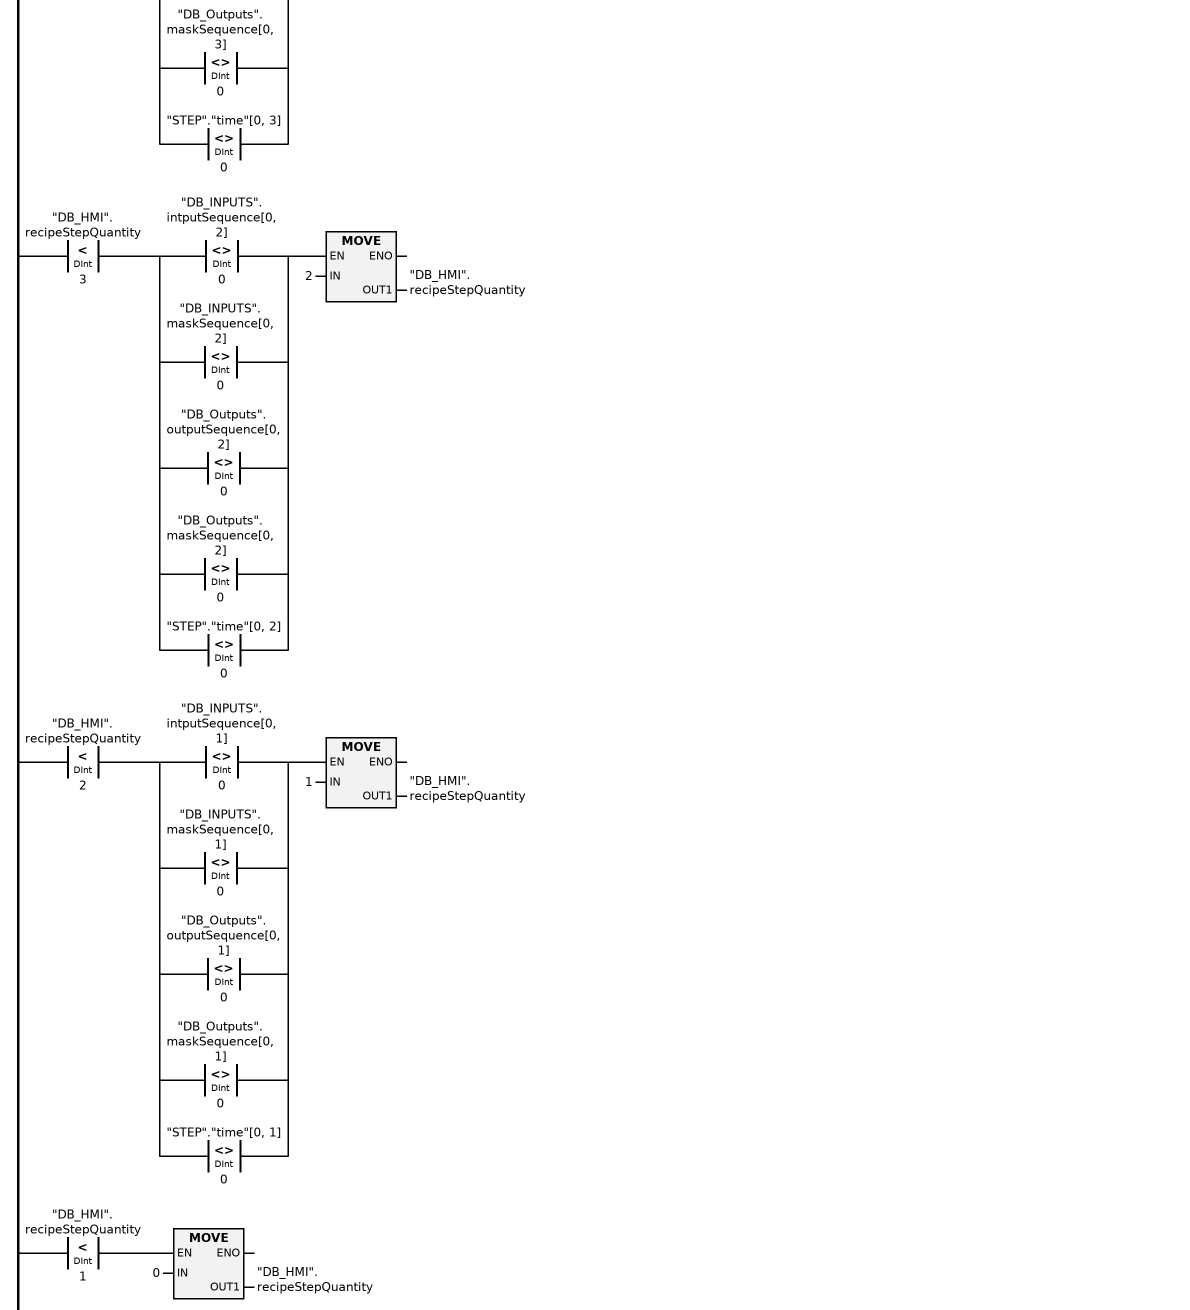
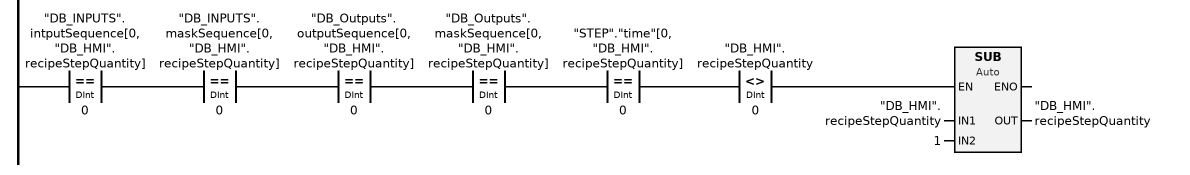
   RUNG wire#powerrail
      { S7_Templates := "SrcType := DInt" } NE_Contact(in1 := "DB_INPUTS".intputSequence[0, 25], in2 := 0)
      wire#w1
      Move(in := 25, out1 => "DB_HMI".recipeStepQuantity)
   END_RUNG
   RUNG wire#powerrail
      { S7_Templates := "SrcType := DInt" } NE_Contact(in1 := "DB_INPUTS".maskSequence[0, 25], in2 := 0)
   END_RUNG wire#w1
   RUNG wire#powerrail
      { S7_Templates := "SrcType := DInt" } NE_Contact(in1 := "DB_Outputs".outputSequence[0, 25], in2 := 0)
   END_RUNG wire#w1
   RUNG wire#powerrail
      { S7_Templates := "SrcType := DInt" } NE_Contact(in1 := "DB_Outputs".maskSequence[0, 25], in2 := 0)
   END_RUNG wire#w1
   RUNG wire#powerrail
      { S7_Templates := "SrcType := DInt" } NE_Contact(in1 := "STEP"."time"[0, 25], in2 := 0)
   END_RUNG wire#w1
   RUNG wire#powerrail
      { S7_Templates := "SrcType := DInt" } LT_Contact(in1 := "DB_HMI".recipeStepQuantity, in2 := 25)
      wire#w2
      { S7_Templates := "SrcType := DInt" } NE_Contact(in1 := "DB_INPUTS".intputSequence[0, 24], in2 := 0)
      wire#w3
      Move(in := 24, out1 => "DB_HMI".recipeStepQuantity)
   END_RUNG
   RUNG wire#w2
      { S7_Templates := "SrcType := DInt" } NE_Contact(in1 := "DB_INPUTS".maskSequence[0, 24], in2 := 0)
   END_RUNG wire#w3
   RUNG wire#w2
      { S7_Templates := "SrcType := DInt" } NE_Contact(in1 := "DB_Outputs".outputSequence[0, 24], in2 := 0)
   END_RUNG wire#w3
   RUNG wire#w2
      { S7_Templates := "SrcType := DInt" } NE_Contact(in1 := "DB_Outputs".maskSequence[0, 24], in2 := 0)
   END_RUNG wire#w3
   RUNG wire#w2
      { S7_Templates := "SrcType := DInt" } NE_Contact(in1 := "STEP"."time"[0, 24], in2 := 0)
   END_RUNG wire#w3
   RUNG wire#powerrail
      { S7_Templates := "SrcType := DInt" } LT_Contact(in1 := "DB_HMI".recipeStepQuantity, in2 := 24)
      wire#w4
      { S7_Templates := "SrcType := DInt" } NE_Contact(in1 := "DB_INPUTS".intputSequence[0, 23], in2 := 0)
      wire#w5
      Move(in := 23, out1 => "DB_HMI".recipeStepQuantity)
   END_RUNG
   RUNG wire#w4
      { S7_Templates := "SrcType := DInt" } NE_Contact(in1 := "DB_INPUTS".maskSequence[0, 23], in2 := 0)
   END_RUNG wire#w5
   RUNG wire#w4
      { S7_Templates := "SrcType := DInt" } NE_Contact(in1 := "DB_Outputs".outputSequence[0, 23], in2 := 0)
   END_RUNG wire#w5
   RUNG wire#w4
      { S7_Templates := "SrcType := DInt" } NE_Contact(in1 := "DB_Outputs".maskSequence[0, 23], in2 := 0)
   END_RUNG wire#w5
   RUNG wire#w4
      { S7_Templates := "SrcType := DInt" } NE_Contact(in1 := "STEP"."time"[0, 23], in2 := 0)
   END_RUNG wire#w5
   RUNG wire#powerrail
      { S7_Templates := "SrcType := DInt" } LT_Contact(in1 := "DB_HMI".recipeStepQuantity, in2 := 23)
      wire#w6
      { S7_Templates := "SrcType := DInt" } NE_Contact(in1 := "DB_INPUTS".intputSequence[0, 22], in2 := 0)
      wire#w7
      Move(in := 22, out1 => "DB_HMI".recipeStepQuantity)
   END_RUNG
   RUNG wire#w6
      { S7_Templates := "SrcType := DInt" } NE_Contact(in1 := "DB_INPUTS".maskSequence[0, 22], in2 := 0)
   END_RUNG wire#w7
   RUNG wire#w6
      { S7_Templates := "SrcType := DInt" } NE_Contact(in1 := "DB_Outputs".outputSequence[0, 22], in2 := 0)
   END_RUNG wire#w7
   RUNG wire#w6
      { S7_Templates := "SrcType := DInt" } NE_Contact(in1 := "DB_Outputs".maskSequence[0, 22], in2 := 0)
   END_RUNG wire#w7
   RUNG wire#w6
      { S7_Templates := "SrcType := DInt" } NE_Contact(in1 := "STEP"."time"[0, 22], in2 := 0)
   END_RUNG wire#w7
   RUNG wire#powerrail
      { S7_Templates := "SrcType := DInt" } LT_Contact(in1 := "DB_HMI".recipeStepQuantity, in2 := 22)
      wire#w8
      { S7_Templates := "SrcType := DInt" } NE_Contact(in1 := "DB_INPUTS".intputSequence[0, 21], in2 := 0)
      wire#w9
      Move(in := 21, out1 => "DB_HMI".recipeStepQuantity)
   END_RUNG
   RUNG wire#w8
      { S7_Templates := "SrcType := DInt" } NE_Contact(in1 := "DB_INPUTS".maskSequence[0, 21], in2 := 0)
   END_RUNG wire#w9
   RUNG wire#w8
      { S7_Templates := "SrcType := DInt" } NE_Contact(in1 := "DB_Outputs".outputSequence[0, 21], in2 := 0)
   END_RUNG wire#w9
   RUNG wire#w8
      { S7_Templates := "SrcType := DInt" } NE_Contact(in1 := "DB_Outputs".maskSequence[0, 21], in2 := 0)
   END_RUNG wire#w9
   RUNG wire#w8
      { S7_Templates := "SrcType := DInt" } NE_Contact(in1 := "STEP"."time"[0, 21], in2 := 0)
   END_RUNG wire#w9
   RUNG wire#powerrail
      { S7_Templates := "SrcType := DInt" } LT_Contact(in1 := "DB_HMI".recipeStepQuantity, in2 := 21)
      wire#w10
      { S7_Templates := "SrcType := DInt" } NE_Contact(in1 := "DB_INPUTS".intputSequence[0, 20], in2 := 0)
      wire#w11
      Move(in := 20, out1 => "DB_HMI".recipeStepQuantity)
   END_RUNG
   RUNG wire#w10
      { S7_Templates := "SrcType := DInt" } NE_Contact(in1 := "DB_INPUTS".maskSequence[0, 20], in2 := 0)
   END_RUNG wire#w11
   RUNG wire#w10
      { S7_Templates := "SrcType := DInt" } NE_Contact(in1 := "DB_Outputs".outputSequence[0, 20], in2 := 0)
   END_RUNG wire#w11
   RUNG wire#w10
      { S7_Templates := "SrcType := DInt" } NE_Contact(in1 := "DB_Outputs".maskSequence[0, 20], in2 := 0)
   END_RUNG wire#w11
   RUNG wire#w10
      { S7_Templates := "SrcType := DInt" } NE_Contact(in1 := "STEP"."time"[0, 20], in2 := 0)
   END_RUNG wire#w11
   RUNG wire#powerrail
      { S7_Templates := "SrcType := DInt" } LT_Contact(in1 := "DB_HMI".recipeStepQuantity, in2 := 20)
      wire#w12
      { S7_Templates := "SrcType := DInt" } NE_Contact(in1 := "DB_INPUTS".intputSequence[0, 19], in2 := 0)
      wire#w13
      Move(in := 19, out1 => "DB_HMI".recipeStepQuantity)
   END_RUNG
   RUNG wire#w12
      { S7_Templates := "SrcType := DInt" } NE_Contact(in1 := "DB_INPUTS".maskSequence[0, 19], in2 := 0)
   END_RUNG wire#w13
   RUNG wire#w12
      { S7_Templates := "SrcType := DInt" } NE_Contact(in1 := "DB_Outputs".outputSequence[0, 19], in2 := 0)
   END_RUNG wire#w13
   RUNG wire#w12
      { S7_Templates := "SrcType := DInt" } NE_Contact(in1 := "DB_Outputs".maskSequence[0, 19], in2 := 0)
   END_RUNG wire#w13
   RUNG wire#w12
      { S7_Templates := "SrcType := DInt" } NE_Contact(in1 := "STEP"."time"[0, 19], in2 := 0)
   END_RUNG wire#w13
   RUNG wire#powerrail
      { S7_Templates := "SrcType := DInt" } LT_Contact(in1 := "DB_HMI".recipeStepQuantity, in2 := 19)
      wire#w14
      { S7_Templates := "SrcType := DInt" } NE_Contact(in1 := "DB_INPUTS".intputSequence[0, 18], in2 := 0)
      wire#w15
      Move(in := 18, out1 => "DB_HMI".recipeStepQuantity)
   END_RUNG
   RUNG wire#w14
      { S7_Templates := "SrcType := DInt" } NE_Contact(in1 := "DB_INPUTS".maskSequence[0, 18], in2 := 0)
   END_RUNG wire#w15
   RUNG wire#w14
      { S7_Templates := "SrcType := DInt" } NE_Contact(in1 := "DB_Outputs".outputSequence[0, 18], in2 := 0)
   END_RUNG wire#w15
   RUNG wire#w14
      { S7_Templates := "SrcType := DInt" } NE_Contact(in1 := "DB_Outputs".maskSequence[0, 18], in2 := 0)
   END_RUNG wire#w15
   RUNG wire#w14
      { S7_Templates := "SrcType := DInt" } NE_Contact(in1 := "STEP"."time"[0, 18], in2 := 0)
   END_RUNG wire#w15
   RUNG wire#powerrail
      { S7_Templates := "SrcType := DInt" } LT_Contact(in1 := "DB_HMI".recipeStepQuantity, in2 := 18)
      wire#w16
      { S7_Templates := "SrcType := DInt" } NE_Contact(in1 := "DB_INPUTS".intputSequence[0, 17], in2 := 0)
      wire#w17
      Move(in := 17, out1 => "DB_HMI".recipeStepQuantity)
   END_RUNG
   RUNG wire#w16
      { S7_Templates := "SrcType := DInt" } NE_Contact(in1 := "DB_INPUTS".maskSequence[0, 17], in2 := 0)
   END_RUNG wire#w17
   RUNG wire#w16
      { S7_Templates := "SrcType := DInt" } NE_Contact(in1 := "DB_Outputs".outputSequence[0, 17], in2 := 0)
   END_RUNG wire#w17
   RUNG wire#w16
      { S7_Templates := "SrcType := DInt" } NE_Contact(in1 := "DB_Outputs".maskSequence[0, 17], in2 := 0)
   END_RUNG wire#w17
   RUNG wire#w16
      { S7_Templates := "SrcType := DInt" } NE_Contact(in1 := "STEP"."time"[0, 17], in2 := 0)
   END_RUNG wire#w17
   RUNG wire#powerrail
      { S7_Templates := "SrcType := DInt" } LT_Contact(in1 := "DB_HMI".recipeStepQuantity, in2 := 17)
      wire#w18
      { S7_Templates := "SrcType := DInt" } NE_Contact(in1 := "DB_INPUTS".intputSequence[0, 16], in2 := 0)
      wire#w19
      Move(in := 16, out1 => "DB_HMI".recipeStepQuantity)
   END_RUNG
   RUNG wire#w18
      { S7_Templates := "SrcType := DInt" } NE_Contact(in1 := "DB_INPUTS".maskSequence[0, 16], in2 := 0)
   END_RUNG wire#w19
   RUNG wire#w18
      { S7_Templates := "SrcType := DInt" } NE_Contact(in1 := "DB_Outputs".outputSequence[0, 16], in2 := 0)
   END_RUNG wire#w19
   RUNG wire#w18
      { S7_Templates := "SrcType := DInt" } NE_Contact(in1 := "DB_Outputs".maskSequence[0, 16], in2 := 0)
   END_RUNG wire#w19
   RUNG wire#w18
      { S7_Templates := "SrcType := DInt" } NE_Contact(in1 := "STEP"."time"[0, 16], in2 := 0)
   END_RUNG wire#w19
   RUNG wire#powerrail
      { S7_Templates := "SrcType := DInt" } LT_Contact(in1 := "DB_HMI".recipeStepQuantity, in2 := 16)
      wire#w20
      { S7_Templates := "SrcType := DInt" } NE_Contact(in1 := "DB_INPUTS".intputSequence[0, 15], in2 := 0)
      wire#w21
      Move(in := 15, out1 => "DB_HMI".recipeStepQuantity)
   END_RUNG
   RUNG wire#w20
      { S7_Templates := "SrcType := DInt" } NE_Contact(in1 := "DB_INPUTS".maskSequence[0, 15], in2 := 0)
   END_RUNG wire#w21
   RUNG wire#w20
      { S7_Templates := "SrcType := DInt" } NE_Contact(in1 := "DB_Outputs".outputSequence[0, 15], in2 := 0)
   END_RUNG wire#w21
   RUNG wire#w20
      { S7_Templates := "SrcType := DInt" } NE_Contact(in1 := "DB_Outputs".maskSequence[0, 15], in2 := 0)
   END_RUNG wire#w21
   RUNG wire#w20
      { S7_Templates := "SrcType := DInt" } NE_Contact(in1 := "STEP"."time"[0, 15], in2 := 0)
   END_RUNG wire#w21
   RUNG wire#powerrail
      { S7_Templates := "SrcType := DInt" } LT_Contact(in1 := "DB_HMI".recipeStepQuantity, in2 := 15)
      wire#w22
      { S7_Templates := "SrcType := DInt" } NE_Contact(in1 := "DB_INPUTS".intputSequence[0, 14], in2 := 0)
      wire#w23
      Move(in := 14, out1 => "DB_HMI".recipeStepQuantity)
   END_RUNG
   RUNG wire#w22
      { S7_Templates := "SrcType := DInt" } NE_Contact(in1 := "DB_INPUTS".maskSequence[0, 14], in2 := 0)
   END_RUNG wire#w23
   RUNG wire#w22
      { S7_Templates := "SrcType := DInt" } NE_Contact(in1 := "DB_Outputs".outputSequence[0, 14], in2 := 0)
   END_RUNG wire#w23
   RUNG wire#w22
      { S7_Templates := "SrcType := DInt" } NE_Contact(in1 := "DB_Outputs".maskSequence[0, 14], in2 := 0)
   END_RUNG wire#w23
   RUNG wire#w22
      { S7_Templates := "SrcType := DInt" } NE_Contact(in1 := "STEP"."time"[0, 14], in2 := 0)
   END_RUNG wire#w23
   RUNG wire#powerrail
      { S7_Templates := "SrcType := DInt" } LT_Contact(in1 := "DB_HMI".recipeStepQuantity, in2 := 14)
      wire#w24
      { S7_Templates := "SrcType := DInt" } NE_Contact(in1 := "DB_INPUTS".intputSequence[0, 13], in2 := 0)
      wire#w25
      Move(in := 13, out1 => "DB_HMI".recipeStepQuantity)
   END_RUNG
   RUNG wire#w24
      { S7_Templates := "SrcType := DInt" } NE_Contact(in1 := "DB_INPUTS".maskSequence[0, 13], in2 := 0)
   END_RUNG wire#w25
   RUNG wire#w24
      { S7_Templates := "SrcType := DInt" } NE_Contact(in1 := "DB_Outputs".outputSequence[0, 13], in2 := 0)
   END_RUNG wire#w25
   RUNG wire#w24
      { S7_Templates := "SrcType := DInt" } NE_Contact(in1 := "DB_Outputs".maskSequence[0, 13], in2 := 0)
   END_RUNG wire#w25
   RUNG wire#w24
      { S7_Templates := "SrcType := DInt" } NE_Contact(in1 := "STEP"."time"[0, 13], in2 := 0)
   END_RUNG wire#w25
   RUNG wire#powerrail
      { S7_Templates := "SrcType := DInt" } LT_Contact(in1 := "DB_HMI".recipeStepQuantity, in2 := 13)
      wire#w26
      { S7_Templates := "SrcType := DInt" } NE_Contact(in1 := "DB_INPUTS".intputSequence[0, 12], in2 := 0)
      wire#w27
      Move(in := 12, out1 => "DB_HMI".recipeStepQuantity)
   END_RUNG
   RUNG wire#w26
      { S7_Templates := "SrcType := DInt" } NE_Contact(in1 := "DB_INPUTS".maskSequence[0, 12], in2 := 0)
   END_RUNG wire#w27
   RUNG wire#w26
      { S7_Templates := "SrcType := DInt" } NE_Contact(in1 := "DB_Outputs".outputSequence[0, 12], in2 := 0)
   END_RUNG wire#w27
   RUNG wire#w26
      { S7_Templates := "SrcType := DInt" } NE_Contact(in1 := "DB_Outputs".maskSequence[0, 12], in2 := 0)
   END_RUNG wire#w27
   RUNG wire#w26
      { S7_Templates := "SrcType := DInt" } NE_Contact(in1 := "STEP"."time"[0, 12], in2 := 0)
   END_RUNG wire#w27
   RUNG wire#powerrail
      { S7_Templates := "SrcType := DInt" } LT_Contact(in1 := "DB_HMI".recipeStepQuantity, in2 := 12)
      wire#w28
      { S7_Templates := "SrcType := DInt" } NE_Contact(in1 := "DB_INPUTS".intputSequence[0, 11], in2 := 0)
      wire#w29
      Move(in := 11, out1 => "DB_HMI".recipeStepQuantity)
   END_RUNG
   RUNG wire#w28
      { S7_Templates := "SrcType := DInt" } NE_Contact(in1 := "DB_INPUTS".maskSequence[0, 11], in2 := 0)
   END_RUNG wire#w29
   RUNG wire#w28
      { S7_Templates := "SrcType := DInt" } NE_Contact(in1 := "DB_Outputs".outputSequence[0, 11], in2 := 0)
   END_RUNG wire#w29
   RUNG wire#w28
      { S7_Templates := "SrcType := DInt" } NE_Contact(in1 := "DB_Outputs".maskSequence[0, 11], in2 := 0)
   END_RUNG wire#w29
   RUNG wire#w28
      { S7_Templates := "SrcType := DInt" } NE_Contact(in1 := "STEP"."time"[0, 11], in2 := 0)
   END_RUNG wire#w29
   RUNG wire#powerrail
      { S7_Templates := "SrcType := DInt" } LT_Contact(in1 := "DB_HMI".recipeStepQuantity, in2 := 11)
      wire#w30
      { S7_Templates := "SrcType := DInt" } NE_Contact(in1 := "DB_INPUTS".intputSequence[0, 10], in2 := 0)
      wire#w31
      Move(in := 10, out1 => "DB_HMI".recipeStepQuantity)
   END_RUNG
   RUNG wire#w30
      { S7_Templates := "SrcType := DInt" } NE_Contact(in1 := "DB_INPUTS".maskSequence[0, 10], in2 := 0)
   END_RUNG wire#w31
   RUNG wire#w30
      { S7_Templates := "SrcType := DInt" } NE_Contact(in1 := "DB_Outputs".outputSequence[0, 10], in2 := 0)
   END_RUNG wire#w31
   RUNG wire#w30
      { S7_Templates := "SrcType := DInt" } NE_Contact(in1 := "DB_Outputs".maskSequence[0, 10], in2 := 0)
   END_RUNG wire#w31
   RUNG wire#w30
      { S7_Templates := "SrcType := DInt" } NE_Contact(in1 := "STEP"."time"[0, 10], in2 := 0)
   END_RUNG wire#w31
   RUNG wire#powerrail
      { S7_Templates := "SrcType := DInt" } LT_Contact(in1 := "DB_HMI".recipeStepQuantity, in2 := 10)
      wire#w32
      { S7_Templates := "SrcType := DInt" } NE_Contact(in1 := "DB_INPUTS".intputSequence[0, 9], in2 := 0)
      wire#w33
      Move(in := 9, out1 => "DB_HMI".recipeStepQuantity)
   END_RUNG
   RUNG wire#w32
      { S7_Templates := "SrcType := DInt" } NE_Contact(in1 := "DB_INPUTS".maskSequence[0, 9], in2 := 0)
   END_RUNG wire#w33
   RUNG wire#w32
      { S7_Templates := "SrcType := DInt" } NE_Contact(in1 := "DB_Outputs".outputSequence[0, 9], in2 := 0)
   END_RUNG wire#w33
   RUNG wire#w32
      { S7_Templates := "SrcType := DInt" } NE_Contact(in1 := "DB_Outputs".maskSequence[0, 9], in2 := 0)
   END_RUNG wire#w33
   RUNG wire#w32
      { S7_Templates := "SrcType := DInt" } NE_Contact(in1 := "STEP"."time"[0, 9], in2 := 0)
   END_RUNG wire#w33
   RUNG wire#powerrail
      { S7_Templates := "SrcType := DInt" } LT_Contact(in1 := "DB_HMI".recipeStepQuantity, in2 := 9)
      wire#w34
      { S7_Templates := "SrcType := DInt" } NE_Contact(in1 := "DB_INPUTS".intputSequence[0, 8], in2 := 0)
      wire#w35
      Move(in := 8, out1 => "DB_HMI".recipeStepQuantity)
   END_RUNG
   RUNG wire#w34
      { S7_Templates := "SrcType := DInt" } NE_Contact(in1 := "DB_INPUTS".maskSequence[0, 8], in2 := 0)
   END_RUNG wire#w35
   RUNG wire#w34
      { S7_Templates := "SrcType := DInt" } NE_Contact(in1 := "DB_Outputs".outputSequence[0, 8], in2 := 0)
   END_RUNG wire#w35
   RUNG wire#w34
      { S7_Templates := "SrcType := DInt" } NE_Contact(in1 := "DB_Outputs".maskSequence[0, 8], in2 := 0)
   END_RUNG wire#w35
   RUNG wire#w34
      { S7_Templates := "SrcType := DInt" } NE_Contact(in1 := "STEP"."time"[0, 8], in2 := 0)
   END_RUNG wire#w35
   RUNG wire#powerrail
      { S7_Templates := "SrcType := DInt" } LT_Contact(in1 := "DB_HMI".recipeStepQuantity, in2 := 8)
      wire#w36
      { S7_Templates := "SrcType := DInt" } NE_Contact(in1 := "DB_INPUTS".intputSequence[0, 7], in2 := 0)
      wire#w37
      Move(in := 7, out1 => "DB_HMI".recipeStepQuantity)
   END_RUNG
   RUNG wire#w36
      { S7_Templates := "SrcType := DInt" } NE_Contact(in1 := "DB_INPUTS".maskSequence[0, 7], in2 := 0)
   END_RUNG wire#w37
   RUNG wire#w36
      { S7_Templates := "SrcType := DInt" } NE_Contact(in1 := "DB_Outputs".outputSequence[0, 7], in2 := 0)
   END_RUNG wire#w37
   RUNG wire#w36
      { S7_Templates := "SrcType := DInt" } NE_Contact(in1 := "DB_Outputs".maskSequence[0, 7], in2 := 0)
   END_RUNG wire#w37
   RUNG wire#w36
      { S7_Templates := "SrcType := DInt" } NE_Contact(in1 := "STEP"."time"[0, 7], in2 := 0)
   END_RUNG wire#w37
   RUNG wire#powerrail
      { S7_Templates := "SrcType := DInt" } LT_Contact(in1 := "DB_HMI".recipeStepQuantity, in2 := 7)
      wire#w38
      { S7_Templates := "SrcType := DInt" } NE_Contact(in1 := "DB_INPUTS".intputSequence[0, 6], in2 := 0)
      wire#w39
      Move(in := 6, out1 => "DB_HMI".recipeStepQuantity)
   END_RUNG
   RUNG wire#w38
      { S7_Templates := "SrcType := DInt" } NE_Contact(in1 := "DB_INPUTS".maskSequence[0, 6], in2 := 0)
   END_RUNG wire#w39
   RUNG wire#w38
      { S7_Templates := "SrcType := DInt" } NE_Contact(in1 := "DB_Outputs".outputSequence[0, 6], in2 := 0)
   END_RUNG wire#w39
   RUNG wire#w38
      { S7_Templates := "SrcType := DInt" } NE_Contact(in1 := "DB_Outputs".maskSequence[0, 6], in2 := 0)
   END_RUNG wire#w39
   RUNG wire#w38
      { S7_Templates := "SrcType := DInt" } NE_Contact(in1 := "STEP"."time"[0, 6], in2 := 0)
   END_RUNG wire#w39
   RUNG wire#powerrail
      { S7_Templates := "SrcType := DInt" } LT_Contact(in1 := "DB_HMI".recipeStepQuantity, in2 := 6)
      wire#w40
      { S7_Templates := "SrcType := DInt" } NE_Contact(in1 := "DB_INPUTS".intputSequence[0, 5], in2 := 0)
      wire#w41
      Move(in := 5, out1 => "DB_HMI".recipeStepQuantity)
   END_RUNG
   RUNG wire#w40
      { S7_Templates := "SrcType := DInt" } NE_Contact(in1 := "DB_INPUTS".maskSequence[0, 5], in2 := 0)
   END_RUNG wire#w41
   RUNG wire#w40
      { S7_Templates := "SrcType := DInt" } NE_Contact(in1 := "DB_Outputs".outputSequence[0, 5], in2 := 0)
   END_RUNG wire#w41
   RUNG wire#w40
      { S7_Templates := "SrcType := DInt" } NE_Contact(in1 := "DB_Outputs".maskSequence[0, 5], in2 := 0)
   END_RUNG wire#w41
   RUNG wire#w40
      { S7_Templates := "SrcType := DInt" } NE_Contact(in1 := "STEP"."time"[0, 5], in2 := 0)
   END_RUNG wire#w41
   RUNG wire#powerrail
      { S7_Templates := "SrcType := DInt" } LT_Contact(in1 := "DB_HMI".recipeStepQuantity, in2 := 5)
      wire#w42
      { S7_Templates := "SrcType := DInt" } NE_Contact(in1 := "DB_INPUTS".intputSequence[0, 4], in2 := 0)
      wire#w43
      Move(in := 4, out1 => "DB_HMI".recipeStepQuantity)
   END_RUNG
   RUNG wire#w42
      { S7_Templates := "SrcType := DInt" } NE_Contact(in1 := "DB_INPUTS".maskSequence[0, 4], in2 := 0)
   END_RUNG wire#w43
   RUNG wire#w42
      { S7_Templates := "SrcType := DInt" } NE_Contact(in1 := "DB_Outputs".outputSequence[0, 4], in2 := 0)
   END_RUNG wire#w43
   RUNG wire#w42
      { S7_Templates := "SrcType := DInt" } NE_Contact(in1 := "DB_Outputs".maskSequence[0, 4], in2 := 0)
   END_RUNG wire#w43
   RUNG wire#w42
      { S7_Templates := "SrcType := DInt" } NE_Contact(in1 := "STEP"."time"[0, 4], in2 := 0)
   END_RUNG wire#w43
   RUNG wire#powerrail
      { S7_Templates := "SrcType := DInt" } LT_Contact(in1 := "DB_HMI".recipeStepQuantity, in2 := 4)
      wire#w44
      { S7_Templates := "SrcType := DInt" } NE_Contact(in1 := "DB_INPUTS".intputSequence[0, 3], in2 := 0)
      wire#w45
      Move(in := 3, out1 => "DB_HMI".recipeStepQuantity)
   END_RUNG
   RUNG wire#w44
      { S7_Templates := "SrcType := DInt" } NE_Contact(in1 := "DB_INPUTS".maskSequence[0, 3], in2 := 0)
   END_RUNG wire#w45
   RUNG wire#w44
      { S7_Templates := "SrcType := DInt" } NE_Contact(in1 := "DB_Outputs".outputSequence[0, 3], in2 := 0)
   END_RUNG wire#w45
   RUNG wire#w44
      { S7_Templates := "SrcType := DInt" } NE_Contact(in1 := "DB_Outputs".maskSequence[0, 3], in2 := 0)
   END_RUNG wire#w45
   RUNG wire#w44
      { S7_Templates := "SrcType := DInt" } NE_Contact(in1 := "STEP"."time"[0, 3], in2 := 0)
   END_RUNG wire#w45
   RUNG wire#powerrail
      { S7_Templates := "SrcType := DInt" } LT_Contact(in1 := "DB_HMI".recipeStepQuantity, in2 := 3)
      wire#w46
      { S7_Templates := "SrcType := DInt" } NE_Contact(in1 := "DB_INPUTS".intputSequence[0, 2], in2 := 0)
      wire#w47
      Move(in := 2, out1 => "DB_HMI".recipeStepQuantity)
   END_RUNG
   RUNG wire#w46
      { S7_Templates := "SrcType := DInt" } NE_Contact(in1 := "DB_INPUTS".maskSequence[0, 2], in2 := 0)
   END_RUNG wire#w47
   RUNG wire#w46
      { S7_Templates := "SrcType := DInt" } NE_Contact(in1 := "DB_Outputs".outputSequence[0, 2], in2 := 0)
   END_RUNG wire#w47
   RUNG wire#w46
      { S7_Templates := "SrcType := DInt" } NE_Contact(in1 := "DB_Outputs".maskSequence[0, 2], in2 := 0)
   END_RUNG wire#w47
   RUNG wire#w46
      { S7_Templates := "SrcType := DInt" } NE_Contact(in1 := "STEP"."time"[0, 2], in2 := 0)
   END_RUNG wire#w47
   RUNG wire#powerrail
      { S7_Templates := "SrcType := DInt" } LT_Contact(in1 := "DB_HMI".recipeStepQuantity, in2 := 2)
      wire#w48
      { S7_Templates := "SrcType := DInt" } NE_Contact(in1 := "DB_INPUTS".intputSequence[0, 1], in2 := 0)
      wire#w49
      Move(in := 1, out1 => "DB_HMI".recipeStepQuantity)
   END_RUNG
   RUNG wire#w48
      { S7_Templates := "SrcType := DInt" } NE_Contact(in1 := "DB_INPUTS".maskSequence[0, 1], in2 := 0)
   END_RUNG wire#w49
   RUNG wire#w48
      { S7_Templates := "SrcType := DInt" } NE_Contact(in1 := "DB_Outputs".outputSequence[0, 1], in2 := 0)
   END_RUNG wire#w49
   RUNG wire#w48
      { S7_Templates := "SrcType := DInt" } NE_Contact(in1 := "DB_Outputs".maskSequence[0, 1], in2 := 0)
   END_RUNG wire#w49
   RUNG wire#w48
      { S7_Templates := "SrcType := DInt" } NE_Contact(in1 := "STEP"."time"[0, 1], in2 := 0)
   END_RUNG wire#w49
   RUNG wire#powerrail
      { S7_Templates := "SrcType := DInt" } LT_Contact(in1 := "DB_HMI".recipeStepQuantity, in2 := 1)
      Move(in := 0, out1 => "DB_HMI".recipeStepQuantity)
   END_RUNG
   RUNG wire#powerrail
      { S7_Templates := "SrcType := DInt" } EQ_Contact(in1 := "DB_INPUTS".intputSequence[0, "DB_HMI".recipeStepQuantity], in2 := 0)
      { S7_Templates := "SrcType := DInt" } EQ_Contact(in1 := "DB_INPUTS".maskSequence[0, "DB_HMI".recipeStepQuantity], in2 := 0)
      { S7_Templates := "SrcType := DInt" } EQ_Contact(in1 := "DB_Outputs".outputSequence[0, "DB_HMI".recipeStepQuantity], in2 := 0)
      { S7_Templates := "SrcType := DInt" } EQ_Contact(in1 := "DB_Outputs".maskSequence[0, "DB_HMI".recipeStepQuantity], in2 := 0)
      { S7_Templates := "SrcType := DInt" } EQ_Contact(in1 := "STEP"."time"[0, "DB_HMI".recipeStepQuantity], in2 := 0)
      { S7_Templates := "SrcType := DInt" } NE_Contact(in1 := "DB_HMI".recipeStepQuantity, in2 := 0)
      Sub(in1 := "DB_HMI".recipeStepQuantity, in2 := 1, out => "DB_HMI".recipeStepQuantity)
   END_RUNG
   // the same network as SCL:
   IF ("DB_INPUTS".intputSequence[0, 25] <> 0) OR ("DB_INPUTS".maskSequence[0, 25] <> 0) OR ("DB_Outputs".outputSequence[0, 25] <> 0) OR ("DB_Outputs".maskSequence[0, 25] <> 0) OR ("STEP"."time"[0, 25] <> 0) THEN
       "DB_HMI".recipeStepQuantity := 25;
   END_IF;
   IF ("DB_HMI".recipeStepQuantity < 25) AND (("DB_INPUTS".intputSequence[0, 24] <> 0) OR ("DB_INPUTS".maskSequence[0, 24] <> 0) OR ("DB_Outputs".outputSequence[0, 24] <> 0) OR ("DB_Outputs".maskSequence[0, 24] <> 0) OR ("STEP"."time"[0, 24] <> 0)) THEN
       "DB_HMI".recipeStepQuantity := 24;
   END_IF;
   IF ("DB_HMI".recipeStepQuantity < 24) AND (("DB_INPUTS".intputSequence[0, 23] <> 0) OR ("DB_INPUTS".maskSequence[0, 23] <> 0) OR ("DB_Outputs".outputSequence[0, 23] <> 0) OR ("DB_Outputs".maskSequence[0, 23] <> 0) OR ("STEP"."time"[0, 23] <> 0)) THEN
       "DB_HMI".recipeStepQuantity := 23;
   END_IF;
   IF ("DB_HMI".recipeStepQuantity < 23) AND (("DB_INPUTS".intputSequence[0, 22] <> 0) OR ("DB_INPUTS".maskSequence[0, 22] <> 0) OR ("DB_Outputs".outputSequence[0, 22] <> 0) OR ("DB_Outputs".maskSequence[0, 22] <> 0) OR ("STEP"."time"[0, 22] <> 0)) THEN
       "DB_HMI".recipeStepQuantity := 22;
   END_IF;
   IF ("DB_HMI".recipeStepQuantity < 22) AND (("DB_INPUTS".intputSequence[0, 21] <> 0) OR ("DB_INPUTS".maskSequence[0, 21] <> 0) OR ("DB_Outputs".outputSequence[0, 21] <> 0) OR ("DB_Outputs".maskSequence[0, 21] <> 0) OR ("STEP"."time"[0, 21] <> 0)) THEN
       "DB_HMI".recipeStepQuantity := 21;
   END_IF;
   IF ("DB_HMI".recipeStepQuantity < 21) AND (("DB_INPUTS".intputSequence[0, 20] <> 0) OR ("DB_INPUTS".maskSequence[0, 20] <> 0) OR ("DB_Outputs".outputSequence[0, 20] <> 0) OR ("DB_Outputs".maskSequence[0, 20] <> 0) OR ("STEP"."time"[0, 20] <> 0)) THEN
       "DB_HMI".recipeStepQuantity := 20;
   END_IF;
   IF ("DB_HMI".recipeStepQuantity < 20) AND (("DB_INPUTS".intputSequence[0, 19] <> 0) OR ("DB_INPUTS".maskSequence[0, 19] <> 0) OR ("DB_Outputs".outputSequence[0, 19] <> 0) OR ("DB_Outputs".maskSequence[0, 19] <> 0) OR ("STEP"."time"[0, 19] <> 0)) THEN
       "DB_HMI".recipeStepQuantity := 19;
   END_IF;
   IF ("DB_HMI".recipeStepQuantity < 19) AND (("DB_INPUTS".intputSequence[0, 18] <> 0) OR ("DB_INPUTS".maskSequence[0, 18] <> 0) OR ("DB_Outputs".outputSequence[0, 18] <> 0) OR ("DB_Outputs".maskSequence[0, 18] <> 0) OR ("STEP"."time"[0, 18] <> 0)) THEN
       "DB_HMI".recipeStepQuantity := 18;
   END_IF;
   IF ("DB_HMI".recipeStepQuantity < 18) AND (("DB_INPUTS".intputSequence[0, 17] <> 0) OR ("DB_INPUTS".maskSequence[0, 17] <> 0) OR ("DB_Outputs".outputSequence[0, 17] <> 0) OR ("DB_Outputs".maskSequence[0, 17] <> 0) OR ("STEP"."time"[0, 17] <> 0)) THEN
       "DB_HMI".recipeStepQuantity := 17;
   END_IF;
   IF ("DB_HMI".recipeStepQuantity < 17) AND (("DB_INPUTS".intputSequence[0, 16] <> 0) OR ("DB_INPUTS".maskSequence[0, 16] <> 0) OR ("DB_Outputs".outputSequence[0, 16] <> 0) OR ("DB_Outputs".maskSequence[0, 16] <> 0) OR ("STEP"."time"[0, 16] <> 0)) THEN
       "DB_HMI".recipeStepQuantity := 16;
   END_IF;
   IF ("DB_HMI".recipeStepQuantity < 16) AND (("DB_INPUTS".intputSequence[0, 15] <> 0) OR ("DB_INPUTS".maskSequence[0, 15] <> 0) OR ("DB_Outputs".outputSequence[0, 15] <> 0) OR ("DB_Outputs".maskSequence[0, 15] <> 0) OR ("STEP"."time"[0, 15] <> 0)) THEN
       "DB_HMI".recipeStepQuantity := 15;
   END_IF;
   IF ("DB_HMI".recipeStepQuantity < 15) AND (("DB_INPUTS".intputSequence[0, 14] <> 0) OR ("DB_INPUTS".maskSequence[0, 14] <> 0) OR ("DB_Outputs".outputSequence[0, 14] <> 0) OR ("DB_Outputs".maskSequence[0, 14] <> 0) OR ("STEP"."time"[0, 14] <> 0)) THEN
       "DB_HMI".recipeStepQuantity := 14;
   END_IF;
   IF ("DB_HMI".recipeStepQuantity < 14) AND (("DB_INPUTS".intputSequence[0, 13] <> 0) OR ("DB_INPUTS".maskSequence[0, 13] <> 0) OR ("DB_Outputs".outputSequence[0, 13] <> 0) OR ("DB_Outputs".maskSequence[0, 13] <> 0) OR ("STEP"."time"[0, 13] <> 0)) THEN
       "DB_HMI".recipeStepQuantity := 13;
   END_IF;
   IF ("DB_HMI".recipeStepQuantity < 13) AND (("DB_INPUTS".intputSequence[0, 12] <> 0) OR ("DB_INPUTS".maskSequence[0, 12] <> 0) OR ("DB_Outputs".outputSequence[0, 12] <> 0) OR ("DB_Outputs".maskSequence[0, 12] <> 0) OR ("STEP"."time"[0, 12] <> 0)) THEN
       "DB_HMI".recipeStepQuantity := 12;
   END_IF;
   IF ("DB_HMI".recipeStepQuantity < 12) AND (("DB_INPUTS".intputSequence[0, 11] <> 0) OR ("DB_INPUTS".maskSequence[0, 11] <> 0) OR ("DB_Outputs".outputSequence[0, 11] <> 0) OR ("DB_Outputs".maskSequence[0, 11] <> 0) OR ("STEP"."time"[0, 11] <> 0)) THEN
       "DB_HMI".recipeStepQuantity := 11;
   END_IF;
   IF ("DB_HMI".recipeStepQuantity < 11) AND (("DB_INPUTS".intputSequence[0, 10] <> 0) OR ("DB_INPUTS".maskSequence[0, 10] <> 0) OR ("DB_Outputs".outputSequence[0, 10] <> 0) OR ("DB_Outputs".maskSequence[0, 10] <> 0) OR ("STEP"."time"[0, 10] <> 0)) THEN
       "DB_HMI".recipeStepQuantity := 10;
   END_IF;
   IF ("DB_HMI".recipeStepQuantity < 10) AND (("DB_INPUTS".intputSequence[0, 9] <> 0) OR ("DB_INPUTS".maskSequence[0, 9] <> 0) OR ("DB_Outputs".outputSequence[0, 9] <> 0) OR ("DB_Outputs".maskSequence[0, 9] <> 0) OR ("STEP"."time"[0, 9] <> 0)) THEN
       "DB_HMI".recipeStepQuantity := 9;
   END_IF;
   IF ("DB_HMI".recipeStepQuantity < 9) AND (("DB_INPUTS".intputSequence[0, 8] <> 0) OR ("DB_INPUTS".maskSequence[0, 8] <> 0) OR ("DB_Outputs".outputSequence[0, 8] <> 0) OR ("DB_Outputs".maskSequence[0, 8] <> 0) OR ("STEP"."time"[0, 8] <> 0)) THEN
       "DB_HMI".recipeStepQuantity := 8;
   END_IF;
   IF ("DB_HMI".recipeStepQuantity < 8) AND (("DB_INPUTS".intputSequence[0, 7] <> 0) OR ("DB_INPUTS".maskSequence[0, 7] <> 0) OR ("DB_Outputs".outputSequence[0, 7] <> 0) OR ("DB_Outputs".maskSequence[0, 7] <> 0) OR ("STEP"."time"[0, 7] <> 0)) THEN
       "DB_HMI".recipeStepQuantity := 7;
   END_IF;
   IF ("DB_HMI".recipeStepQuantity < 7) AND (("DB_INPUTS".intputSequence[0, 6] <> 0) OR ("DB_INPUTS".maskSequence[0, 6] <> 0) OR ("DB_Outputs".outputSequence[0, 6] <> 0) OR ("DB_Outputs".maskSequence[0, 6] <> 0) OR ("STEP"."time"[0, 6] <> 0)) THEN
       "DB_HMI".recipeStepQuantity := 6;
   END_IF;
   IF ("DB_HMI".recipeStepQuantity < 6) AND (("DB_INPUTS".intputSequence[0, 5] <> 0) OR ("DB_INPUTS".maskSequence[0, 5] <> 0) OR ("DB_Outputs".outputSequence[0, 5] <> 0) OR ("DB_Outputs".maskSequence[0, 5] <> 0) OR ("STEP"."time"[0, 5] <> 0)) THEN
       "DB_HMI".recipeStepQuantity := 5;
   END_IF;
   IF ("DB_HMI".recipeStepQuantity < 5) AND (("DB_INPUTS".intputSequence[0, 4] <> 0) OR ("DB_INPUTS".maskSequence[0, 4] <> 0) OR ("DB_Outputs".outputSequence[0, 4] <> 0) OR ("DB_Outputs".maskSequence[0, 4] <> 0) OR ("STEP"."time"[0, 4] <> 0)) THEN
       "DB_HMI".recipeStepQuantity := 4;
   END_IF;
   IF ("DB_HMI".recipeStepQuantity < 4) AND (("DB_INPUTS".intputSequence[0, 3] <> 0) OR ("DB_INPUTS".maskSequence[0, 3] <> 0) OR ("DB_Outputs".outputSequence[0, 3] <> 0) OR ("DB_Outputs".maskSequence[0, 3] <> 0) OR ("STEP"."time"[0, 3] <> 0)) THEN
       "DB_HMI".recipeStepQuantity := 3;
   END_IF;
   IF ("DB_HMI".recipeStepQuantity < 3) AND (("DB_INPUTS".intputSequence[0, 2] <> 0) OR ("DB_INPUTS".maskSequence[0, 2] <> 0) OR ("DB_Outputs".outputSequence[0, 2] <> 0) OR ("DB_Outputs".maskSequence[0, 2] <> 0) OR ("STEP"."time"[0, 2] <> 0)) THEN
       "DB_HMI".recipeStepQuantity := 2;
   END_IF;
   IF ("DB_HMI".recipeStepQuantity < 2) AND (("DB_INPUTS".intputSequence[0, 1] <> 0) OR ("DB_INPUTS".maskSequence[0, 1] <> 0) OR ("DB_Outputs".outputSequence[0, 1] <> 0) OR ("DB_Outputs".maskSequence[0, 1] <> 0) OR ("STEP"."time"[0, 1] <> 0)) THEN
       "DB_HMI".recipeStepQuantity := 1;
   END_IF;
   IF "DB_HMI".recipeStepQuantity < 1 THEN "DB_HMI".recipeStepQuantity := 0; END_IF;
   IF ("DB_INPUTS".intputSequence[0, "DB_HMI".recipeStepQuantity] = 0) AND ("DB_INPUTS".maskSequence[0, "DB_HMI".recipeStepQuantity] = 0) AND ("DB_Outputs".outputSequence[0, "DB_HMI".recipeStepQuantity] = 0) AND ("DB_Outputs".maskSequence[0, "DB_HMI".recipeStepQuantity] = 0) AND ("STEP"."time"[0, "DB_HMI".recipeStepQuantity] = 0) AND ("DB_HMI".recipeStepQuantity <> 0) THEN
       "DB_HMI".recipeStepQuantity := "DB_HMI".recipeStepQuantity - 1;
   END_IF;
END_REGION

REGION Network 9: INPUT STATUS TO SHOW ON SCREEN
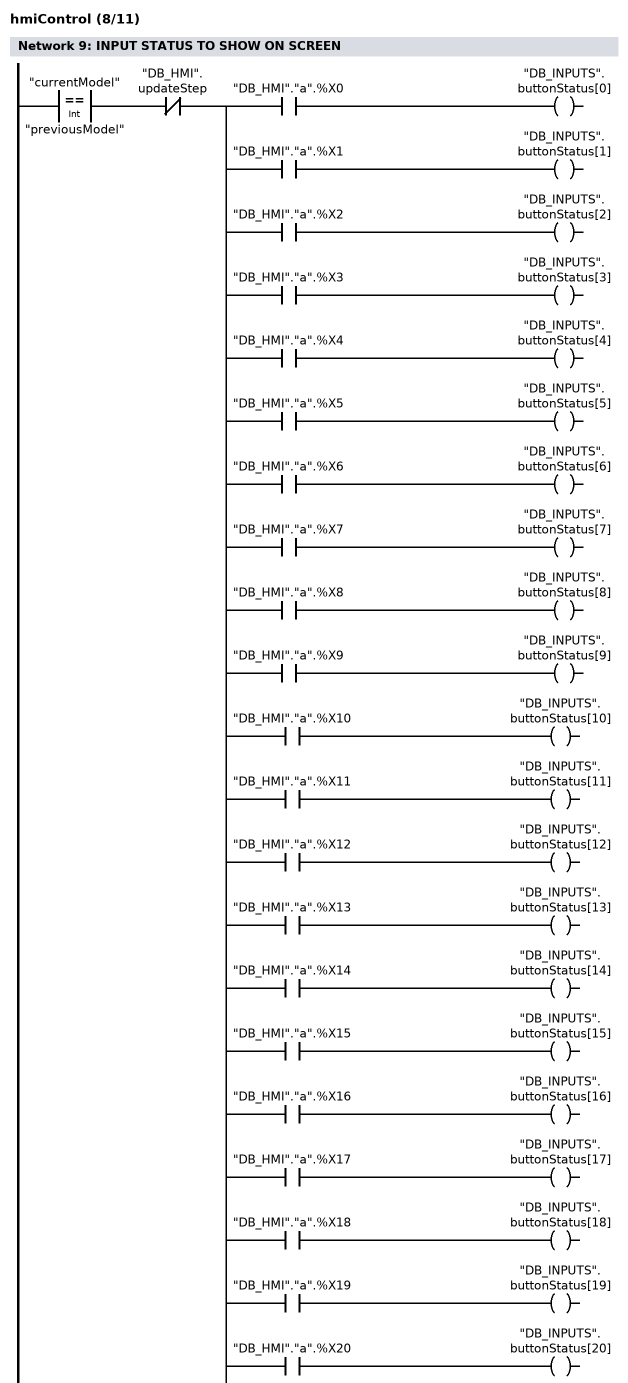
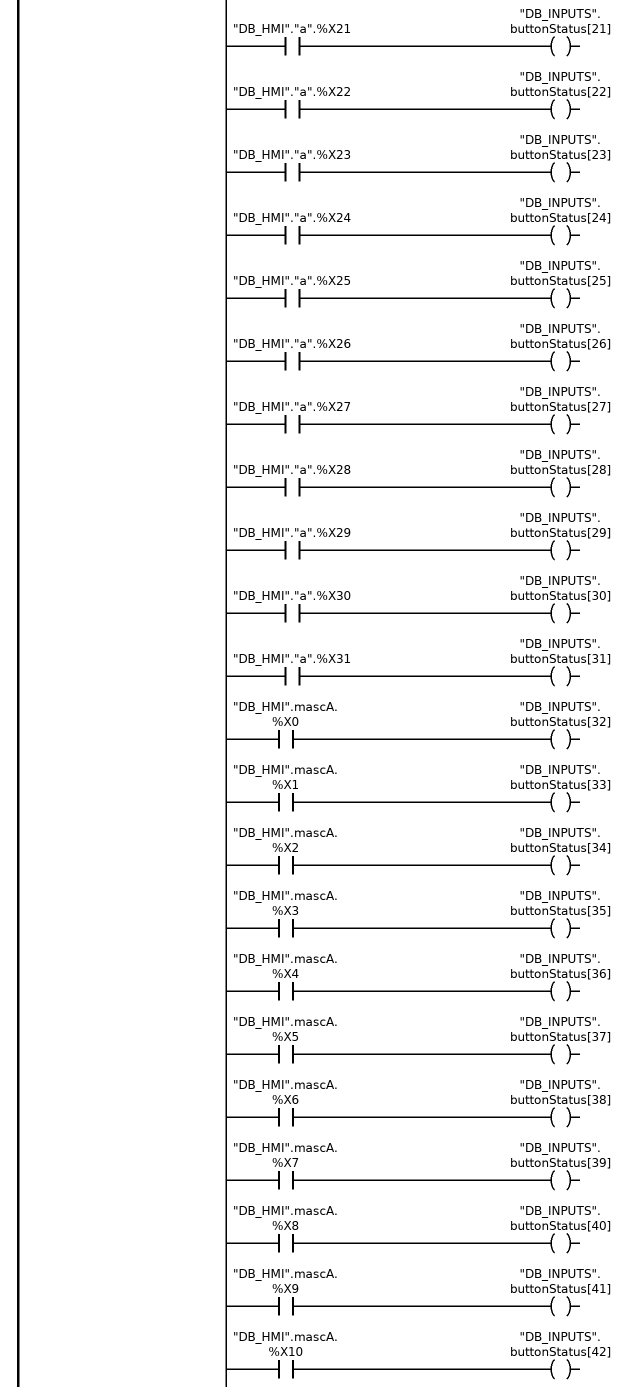
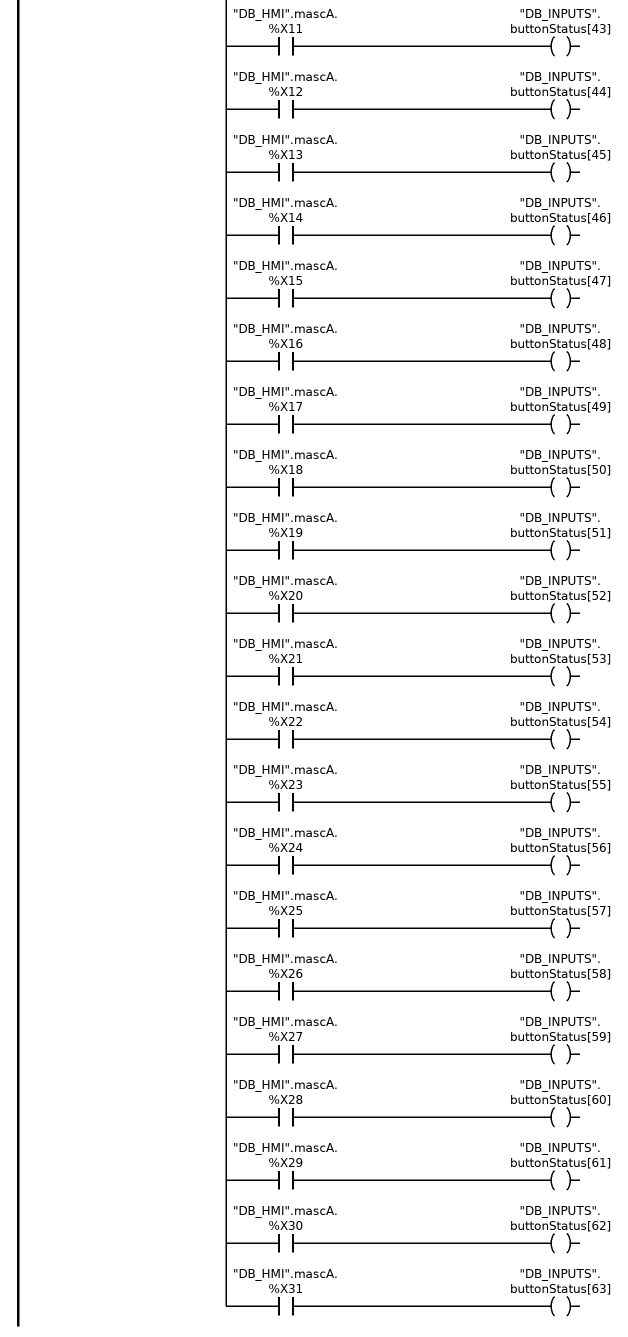
   RUNG wire#powerrail
      { S7_Templates := "SrcType := Int" } EQ_Contact(in1 := "currentModel", in2 := "previousModel")
      I_Contact( "DB_HMI".updateStep )
      wire#w1
      Contact( "DB_HMI"."a".%X0 )
      Coil( "DB_INPUTS".buttonStatus[0] )
   END_RUNG
   RUNG wire#w1
      Contact( "DB_HMI"."a".%X1 )
      Coil( "DB_INPUTS".buttonStatus[1] )
   END_RUNG
   RUNG wire#w1
      Contact( "DB_HMI"."a".%X2 )
      Coil( "DB_INPUTS".buttonStatus[2] )
   END_RUNG
   RUNG wire#w1
      Contact( "DB_HMI"."a".%X3 )
      Coil( "DB_INPUTS".buttonStatus[3] )
   END_RUNG
   RUNG wire#w1
      Contact( "DB_HMI"."a".%X4 )
      Coil( "DB_INPUTS".buttonStatus[4] )
   END_RUNG
   RUNG wire#w1
      Contact( "DB_HMI"."a".%X5 )
      Coil( "DB_INPUTS".buttonStatus[5] )
   END_RUNG
   RUNG wire#w1
      Contact( "DB_HMI"."a".%X6 )
      Coil( "DB_INPUTS".buttonStatus[6] )
   END_RUNG
   RUNG wire#w1
      Contact( "DB_HMI"."a".%X7 )
      Coil( "DB_INPUTS".buttonStatus[7] )
   END_RUNG
   RUNG wire#w1
      Contact( "DB_HMI"."a".%X8 )
      Coil( "DB_INPUTS".buttonStatus[8] )
   END_RUNG
   RUNG wire#w1
      Contact( "DB_HMI"."a".%X9 )
      Coil( "DB_INPUTS".buttonStatus[9] )
   END_RUNG
   RUNG wire#w1
      Contact( "DB_HMI"."a".%X10 )
      Coil( "DB_INPUTS".buttonStatus[10] )
   END_RUNG
   RUNG wire#w1
      Contact( "DB_HMI"."a".%X11 )
      Coil( "DB_INPUTS".buttonStatus[11] )
   END_RUNG
   RUNG wire#w1
      Contact( "DB_HMI"."a".%X12 )
      Coil( "DB_INPUTS".buttonStatus[12] )
   END_RUNG
   RUNG wire#w1
      Contact( "DB_HMI"."a".%X13 )
      Coil( "DB_INPUTS".buttonStatus[13] )
   END_RUNG
   RUNG wire#w1
      Contact( "DB_HMI"."a".%X14 )
      Coil( "DB_INPUTS".buttonStatus[14] )
   END_RUNG
   RUNG wire#w1
      Contact( "DB_HMI"."a".%X15 )
      Coil( "DB_INPUTS".buttonStatus[15] )
   END_RUNG
   RUNG wire#w1
      Contact( "DB_HMI"."a".%X16 )
      Coil( "DB_INPUTS".buttonStatus[16] )
   END_RUNG
   RUNG wire#w1
      Contact( "DB_HMI"."a".%X17 )
      Coil( "DB_INPUTS".buttonStatus[17] )
   END_RUNG
   RUNG wire#w1
      Contact( "DB_HMI"."a".%X18 )
      Coil( "DB_INPUTS".buttonStatus[18] )
   END_RUNG
   RUNG wire#w1
      Contact( "DB_HMI"."a".%X19 )
      Coil( "DB_INPUTS".buttonStatus[19] )
   END_RUNG
   RUNG wire#w1
      Contact( "DB_HMI"."a".%X20 )
      Coil( "DB_INPUTS".buttonStatus[20] )
   END_RUNG
   RUNG wire#w1
      Contact( "DB_HMI"."a".%X21 )
      Coil( "DB_INPUTS".buttonStatus[21] )
   END_RUNG
   RUNG wire#w1
      Contact( "DB_HMI"."a".%X22 )
      Coil( "DB_INPUTS".buttonStatus[22] )
   END_RUNG
   RUNG wire#w1
      Contact( "DB_HMI"."a".%X23 )
      Coil( "DB_INPUTS".buttonStatus[23] )
   END_RUNG
   RUNG wire#w1
      Contact( "DB_HMI"."a".%X24 )
      Coil( "DB_INPUTS".buttonStatus[24] )
   END_RUNG
   RUNG wire#w1
      Contact( "DB_HMI"."a".%X25 )
      Coil( "DB_INPUTS".buttonStatus[25] )
   END_RUNG
   RUNG wire#w1
      Contact( "DB_HMI"."a".%X26 )
      Coil( "DB_INPUTS".buttonStatus[26] )
   END_RUNG
   RUNG wire#w1
      Contact( "DB_HMI"."a".%X27 )
      Coil( "DB_INPUTS".buttonStatus[27] )
   END_RUNG
   RUNG wire#w1
      Contact( "DB_HMI"."a".%X28 )
      Coil( "DB_INPUTS".buttonStatus[28] )
   END_RUNG
   RUNG wire#w1
      Contact( "DB_HMI"."a".%X29 )
      Coil( "DB_INPUTS".buttonStatus[29] )
   END_RUNG
   RUNG wire#w1
      Contact( "DB_HMI"."a".%X30 )
      Coil( "DB_INPUTS".buttonStatus[30] )
   END_RUNG
   RUNG wire#w1
      Contact( "DB_HMI"."a".%X31 )
      Coil( "DB_INPUTS".buttonStatus[31] )
   END_RUNG
   RUNG wire#w1
      Contact( "DB_HMI".mascA.%X0 )
      Coil( "DB_INPUTS".buttonStatus[32] )
   END_RUNG
   RUNG wire#w1
      Contact( "DB_HMI".mascA.%X1 )
      Coil( "DB_INPUTS".buttonStatus[33] )
   END_RUNG
   RUNG wire#w1
      Contact( "DB_HMI".mascA.%X2 )
      Coil( "DB_INPUTS".buttonStatus[34] )
   END_RUNG
   RUNG wire#w1
      Contact( "DB_HMI".mascA.%X3 )
      Coil( "DB_INPUTS".buttonStatus[35] )
   END_RUNG
   RUNG wire#w1
      Contact( "DB_HMI".mascA.%X4 )
      Coil( "DB_INPUTS".buttonStatus[36] )
   END_RUNG
   RUNG wire#w1
      Contact( "DB_HMI".mascA.%X5 )
      Coil( "DB_INPUTS".buttonStatus[37] )
   END_RUNG
   RUNG wire#w1
      Contact( "DB_HMI".mascA.%X6 )
      Coil( "DB_INPUTS".buttonStatus[38] )
   END_RUNG
   RUNG wire#w1
      Contact( "DB_HMI".mascA.%X7 )
      Coil( "DB_INPUTS".buttonStatus[39] )
   END_RUNG
   RUNG wire#w1
      Contact( "DB_HMI".mascA.%X8 )
      Coil( "DB_INPUTS".buttonStatus[40] )
   END_RUNG
   RUNG wire#w1
      Contact( "DB_HMI".mascA.%X9 )
      Coil( "DB_INPUTS".buttonStatus[41] )
   END_RUNG
   RUNG wire#w1
      Contact( "DB_HMI".mascA.%X10 )
      Coil( "DB_INPUTS".buttonStatus[42] )
   END_RUNG
   RUNG wire#w1
      Contact( "DB_HMI".mascA.%X11 )
      Coil( "DB_INPUTS".buttonStatus[43] )
   END_RUNG
   RUNG wire#w1
      Contact( "DB_HMI".mascA.%X12 )
      Coil( "DB_INPUTS".buttonStatus[44] )
   END_RUNG
   RUNG wire#w1
      Contact( "DB_HMI".mascA.%X13 )
      Coil( "DB_INPUTS".buttonStatus[45] )
   END_RUNG
   RUNG wire#w1
      Contact( "DB_HMI".mascA.%X14 )
      Coil( "DB_INPUTS".buttonStatus[46] )
   END_RUNG
   RUNG wire#w1
      Contact( "DB_HMI".mascA.%X15 )
      Coil( "DB_INPUTS".buttonStatus[47] )
   END_RUNG
   RUNG wire#w1
      Contact( "DB_HMI".mascA.%X16 )
      Coil( "DB_INPUTS".buttonStatus[48] )
   END_RUNG
   RUNG wire#w1
      Contact( "DB_HMI".mascA.%X17 )
      Coil( "DB_INPUTS".buttonStatus[49] )
   END_RUNG
   RUNG wire#w1
      Contact( "DB_HMI".mascA.%X18 )
      Coil( "DB_INPUTS".buttonStatus[50] )
   END_RUNG
   RUNG wire#w1
      Contact( "DB_HMI".mascA.%X19 )
      Coil( "DB_INPUTS".buttonStatus[51] )
   END_RUNG
   RUNG wire#w1
      Contact( "DB_HMI".mascA.%X20 )
      Coil( "DB_INPUTS".buttonStatus[52] )
   END_RUNG
   RUNG wire#w1
      Contact( "DB_HMI".mascA.%X21 )
      Coil( "DB_INPUTS".buttonStatus[53] )
   END_RUNG
   RUNG wire#w1
      Contact( "DB_HMI".mascA.%X22 )
      Coil( "DB_INPUTS".buttonStatus[54] )
   END_RUNG
   RUNG wire#w1
      Contact( "DB_HMI".mascA.%X23 )
      Coil( "DB_INPUTS".buttonStatus[55] )
   END_RUNG
   RUNG wire#w1
      Contact( "DB_HMI".mascA.%X24 )
      Coil( "DB_INPUTS".buttonStatus[56] )
   END_RUNG
   RUNG wire#w1
      Contact( "DB_HMI".mascA.%X25 )
      Coil( "DB_INPUTS".buttonStatus[57] )
   END_RUNG
   RUNG wire#w1
      Contact( "DB_HMI".mascA.%X26 )
      Coil( "DB_INPUTS".buttonStatus[58] )
   END_RUNG
   RUNG wire#w1
      Contact( "DB_HMI".mascA.%X27 )
      Coil( "DB_INPUTS".buttonStatus[59] )
   END_RUNG
   RUNG wire#w1
      Contact( "DB_HMI".mascA.%X28 )
      Coil( "DB_INPUTS".buttonStatus[60] )
   END_RUNG
   RUNG wire#w1
      Contact( "DB_HMI".mascA.%X29 )
      Coil( "DB_INPUTS".buttonStatus[61] )
   END_RUNG
   RUNG wire#w1
      Contact( "DB_HMI".mascA.%X30 )
      Coil( "DB_INPUTS".buttonStatus[62] )
   END_RUNG
   RUNG wire#w1
      Contact( "DB_HMI".mascA.%X31 )
      Coil( "DB_INPUTS".buttonStatus[63] )
   END_RUNG
   // the same network as SCL:
   #_w1 := ("currentModel" = "previousModel") AND NOT "DB_HMI".updateStep;
   "DB_INPUTS".buttonStatus[0] := #_w1 AND "DB_HMI"."a".%X0;
   "DB_INPUTS".buttonStatus[1] := #_w1 AND "DB_HMI"."a".%X1;
   "DB_INPUTS".buttonStatus[2] := #_w1 AND "DB_HMI"."a".%X2;
   "DB_INPUTS".buttonStatus[3] := #_w1 AND "DB_HMI"."a".%X3;
   "DB_INPUTS".buttonStatus[4] := #_w1 AND "DB_HMI"."a".%X4;
   "DB_INPUTS".buttonStatus[5] := #_w1 AND "DB_HMI"."a".%X5;
   "DB_INPUTS".buttonStatus[6] := #_w1 AND "DB_HMI"."a".%X6;
   "DB_INPUTS".buttonStatus[7] := #_w1 AND "DB_HMI"."a".%X7;
   "DB_INPUTS".buttonStatus[8] := #_w1 AND "DB_HMI"."a".%X8;
   "DB_INPUTS".buttonStatus[9] := #_w1 AND "DB_HMI"."a".%X9;
   "DB_INPUTS".buttonStatus[10] := #_w1 AND "DB_HMI"."a".%X10;
   "DB_INPUTS".buttonStatus[11] := #_w1 AND "DB_HMI"."a".%X11;
   "DB_INPUTS".buttonStatus[12] := #_w1 AND "DB_HMI"."a".%X12;
   "DB_INPUTS".buttonStatus[13] := #_w1 AND "DB_HMI"."a".%X13;
   "DB_INPUTS".buttonStatus[14] := #_w1 AND "DB_HMI"."a".%X14;
   "DB_INPUTS".buttonStatus[15] := #_w1 AND "DB_HMI"."a".%X15;
   "DB_INPUTS".buttonStatus[16] := #_w1 AND "DB_HMI"."a".%X16;
   "DB_INPUTS".buttonStatus[17] := #_w1 AND "DB_HMI"."a".%X17;
   "DB_INPUTS".buttonStatus[18] := #_w1 AND "DB_HMI"."a".%X18;
   "DB_INPUTS".buttonStatus[19] := #_w1 AND "DB_HMI"."a".%X19;
   "DB_INPUTS".buttonStatus[20] := #_w1 AND "DB_HMI"."a".%X20;
   "DB_INPUTS".buttonStatus[21] := #_w1 AND "DB_HMI"."a".%X21;
   "DB_INPUTS".buttonStatus[22] := #_w1 AND "DB_HMI"."a".%X22;
   "DB_INPUTS".buttonStatus[23] := #_w1 AND "DB_HMI"."a".%X23;
   "DB_INPUTS".buttonStatus[24] := #_w1 AND "DB_HMI"."a".%X24;
   "DB_INPUTS".buttonStatus[25] := #_w1 AND "DB_HMI"."a".%X25;
   "DB_INPUTS".buttonStatus[26] := #_w1 AND "DB_HMI"."a".%X26;
   "DB_INPUTS".buttonStatus[27] := #_w1 AND "DB_HMI"."a".%X27;
   "DB_INPUTS".buttonStatus[28] := #_w1 AND "DB_HMI"."a".%X28;
   "DB_INPUTS".buttonStatus[29] := #_w1 AND "DB_HMI"."a".%X29;
   "DB_INPUTS".buttonStatus[30] := #_w1 AND "DB_HMI"."a".%X30;
   "DB_INPUTS".buttonStatus[31] := #_w1 AND "DB_HMI"."a".%X31;
   "DB_INPUTS".buttonStatus[32] := #_w1 AND "DB_HMI".mascA.%X0;
   "DB_INPUTS".buttonStatus[33] := #_w1 AND "DB_HMI".mascA.%X1;
   "DB_INPUTS".buttonStatus[34] := #_w1 AND "DB_HMI".mascA.%X2;
   "DB_INPUTS".buttonStatus[35] := #_w1 AND "DB_HMI".mascA.%X3;
   "DB_INPUTS".buttonStatus[36] := #_w1 AND "DB_HMI".mascA.%X4;
   "DB_INPUTS".buttonStatus[37] := #_w1 AND "DB_HMI".mascA.%X5;
   "DB_INPUTS".buttonStatus[38] := #_w1 AND "DB_HMI".mascA.%X6;
   "DB_INPUTS".buttonStatus[39] := #_w1 AND "DB_HMI".mascA.%X7;
   "DB_INPUTS".buttonStatus[40] := #_w1 AND "DB_HMI".mascA.%X8;
   "DB_INPUTS".buttonStatus[41] := #_w1 AND "DB_HMI".mascA.%X9;
   "DB_INPUTS".buttonStatus[42] := #_w1 AND "DB_HMI".mascA.%X10;
   "DB_INPUTS".buttonStatus[43] := #_w1 AND "DB_HMI".mascA.%X11;
   "DB_INPUTS".buttonStatus[44] := #_w1 AND "DB_HMI".mascA.%X12;
   "DB_INPUTS".buttonStatus[45] := #_w1 AND "DB_HMI".mascA.%X13;
   "DB_INPUTS".buttonStatus[46] := #_w1 AND "DB_HMI".mascA.%X14;
   "DB_INPUTS".buttonStatus[47] := #_w1 AND "DB_HMI".mascA.%X15;
   "DB_INPUTS".buttonStatus[48] := #_w1 AND "DB_HMI".mascA.%X16;
   "DB_INPUTS".buttonStatus[49] := #_w1 AND "DB_HMI".mascA.%X17;
   "DB_INPUTS".buttonStatus[50] := #_w1 AND "DB_HMI".mascA.%X18;
   "DB_INPUTS".buttonStatus[51] := #_w1 AND "DB_HMI".mascA.%X19;
   "DB_INPUTS".buttonStatus[52] := #_w1 AND "DB_HMI".mascA.%X20;
   "DB_INPUTS".buttonStatus[53] := #_w1 AND "DB_HMI".mascA.%X21;
   "DB_INPUTS".buttonStatus[54] := #_w1 AND "DB_HMI".mascA.%X22;
   "DB_INPUTS".buttonStatus[55] := #_w1 AND "DB_HMI".mascA.%X23;
   "DB_INPUTS".buttonStatus[56] := #_w1 AND "DB_HMI".mascA.%X24;
   "DB_INPUTS".buttonStatus[57] := #_w1 AND "DB_HMI".mascA.%X25;
   "DB_INPUTS".buttonStatus[58] := #_w1 AND "DB_HMI".mascA.%X26;
   "DB_INPUTS".buttonStatus[59] := #_w1 AND "DB_HMI".mascA.%X27;
   "DB_INPUTS".buttonStatus[60] := #_w1 AND "DB_HMI".mascA.%X28;
   "DB_INPUTS".buttonStatus[61] := #_w1 AND "DB_HMI".mascA.%X29;
   "DB_INPUTS".buttonStatus[62] := #_w1 AND "DB_HMI".mascA.%X30;
   "DB_INPUTS".buttonStatus[63] := #_w1 AND "DB_HMI".mascA.%X31;
END_REGION

REGION Network 10: OUTPUT STATUS TO SHOW ON SCREEN
